(* CoDeSys 2.3 project: cy-wg-06-005.pro *)
(* Title: cy-wg-06 - ClevergyAS *)
(* Author: Andrea Ravasio *)
(* Libraries: Standard.lib 2.12.10 13:48:34, Util.lib*26.9.14 10:12:46, Visual.lib 2.12.10 13:48:34, WagoLibIdent.lib 25.2.13 10:12:16, WagoLibStatus.lib 2.12.10 13:48:32, SysLibFile.lib 2.12.10 13:48:34, SysLibRtc.lib 2.12.10 13:48:32, SysLibSockets.lib 10.2.11 08:20:54, SysLibEvent.lib 2.12.10 13:48:34, SysLibPlcCtrl.lib 2.12.10 13:48:32, SysLibCallback.lib 2.12.10 13:48:32, mod_com.lib 2.12.10 13:48:32, SerComm.lib 31.5.11 07:54:36, Serial_Interface_01.lib 22.4.13 11:50:14, Modb_l05.lib*13.5.15 09:30:08, MBus_03.lib 9.2.13 16:51:58 *)

(* PLC configuration (modules and I/O channels)
K-Bus [K_Bus] node 0, in %IB0 out %QB0
  0750-0402 4 DI 24 V DC 3.0ms [Type_1_4_Channels] node 0, in %IB8 out %QB8 {INTTypePAAssignment = PLC; INTTypeModule = plugged}
    VPN_OUT2 AT %IX4.0 [BOOLOnX_I] Ch_1 Digital input
    KEY_QE_ST AT %IX4.1 [BOOLOnX_I] Ch_2 Digital input
    AT %IX4.2 [BOOLOnX_I] Ch_3 Digital input
    AT %IX4.3 [BOOLOnX_I] Ch_4 Digital input
  0750-0504 4 DO 24V DC 0.5A [Type_10_4_Channels] node 1, in %IB8 out %QB8 {INTTypePAAssignment = PLC; INTTypeModule = plugged}
    AT %QX4.0 [BOOLOnX_Q] Ch_1 Digital output
    AT %QX4.1 [BOOLOnX_Q] Ch_2 Digital output
    TEST1 AT %QX4.2 [BOOLOnX_Q] Ch_3 Digital output
    TEST2 AT %QX4.3 [BOOLOnX_Q] Ch_4 Digital output
  0750-0653/0003-0000#03 RS485 Interface (Adjustable), 3 Bytes [Type_21_1_Channels] node 2, in %IB4 out %QB4 {INTTypePAAssignment = PLC; INTTypeModule = plugged}
    AT %IX0.0 [BOOLOnX_I] Transmission acknowledgement
    AT %IX0.1 [BOOLOnX_I] Reception request
    AT %IX0.2 [BOOLOnX_I] Initialization acknowledgement
    AT %IX0.3 [BOOLOnX_I] Input buffer is full
    AT %IX0.4 [BOOLOnX_I] Number of received characters Bit 0
    AT %IX0.5 [BOOLOnX_I] Number of received characters Bit 1
    AT %IX0.6 [BOOLOnX_I] Number of received characters Bit 2
    AT %IB1 [BYTEOnB_I] Input data Byte 0
    AT %IB2 [BYTEOnB_I] Input data Byte 1
    AT %IB3 [BYTEOnB_I] Input data Byte 2
    AT %QX0.0 [BOOLOnX_Q] Transmission request
    AT %QX0.1 [BOOLOnX_Q] Reception acknowledgement
    AT %QX0.2 [BOOLOnX_Q] Initialization request
    AT %QX0.4 [BOOLOnX_Q] Number of characters Bit 0
    AT %QX0.5 [BOOLOnX_Q] Number of characters Bit 1
    AT %QX0.6 [BOOLOnX_Q] Number of characters Bit 2
    AT %QB1 [BYTEOnB_Q] Output data Byte 0
    AT %QB2 [BYTEOnB_Q] Output data Byte 1
    AT %QB3 [BYTEOnB_Q] Output data Byte 2
  0750-0650/0003-0000#03 RS 232 C Interface (Adjustable), 3 Byte [Type_21_1_Channels] node 0, in %IB4 out %QB4 {INTTypePAAssignment = PLC; INTTypeModule = plugged}
    AT %IX2.0 [BOOLOnX_I] Transmission acknowledgement
    AT %IX2.1 [BOOLOnX_I] Reception request
    AT %IX2.2 [BOOLOnX_I] Initialization acknowledgement
    AT %IX2.3 [BOOLOnX_I] Input buffer is full
    AT %IX2.4 [BOOLOnX_I] Number of received characters Bit 0
    AT %IX2.5 [BOOLOnX_I] Number of received characters Bit 1
    AT %IX2.6 [BOOLOnX_I] Number of received characters Bit 2
    AT %IB5 [BYTEOnB_I] Input data Byte 0
    AT %IB6 [BYTEOnB_I] Input data Byte 1
    AT %IB7 [BYTEOnB_I] Input data Byte 2
    AT %QX2.0 [BOOLOnX_Q] Transmission request
    AT %QX2.1 [BOOLOnX_Q] Reception acknowledgement
    AT %QX2.2 [BOOLOnX_Q] Initialization request
    AT %QX2.4 [BOOLOnX_Q] Number of characters Bit 0
    AT %QX2.5 [BOOLOnX_Q] Number of characters Bit 1
    AT %QX2.6 [BOOLOnX_Q] Number of characters Bit 2
    AT %QB5 [BYTEOnB_Q] Output data Byte 0
    AT %QB6 [BYTEOnB_Q] Output data Byte 1
    AT %QB7 [BYTEOnB_Q] Output data Byte 2
Fieldbus variables [FB_VARS] node 1, in %IB0 out %QB0
Flag variables [FLAG_VARS] node 2, in %IB0 out %QB0
Modbus-Master [MB_MASTER] node 3, in %IB0 out %QB0
*)

(* Global variable list: Global_Constants *)
VAR_GLOBAL CONSTANT

	Plant_NAME			: STRING :='cySN:6 cyVER:5 - Gavazzeni D Energetiche';
	Plant_SN			: DWORD  :=6;  		(* S/N Impianto di telecontrollo *)
	Plant_SW_VER		: WORD   :=5;		(* Versione SW installata *)

	(* Parameters *)
	Plant_DefaultTAmb	: INT	:=100;		(* [.1°C] Temperatura ambiente di default in caso di rottura sonda *)
	Plant_MaxRunTAmb	: INT   :=250; 		(* [.1°C] Temperatura ambiente massima funzionamento impianto *)
	Plant_AntiFreezeTAmb: INT   :=-40;		(* [.1°C] Antifreeze temperature, start circulators *)
	Plant_VRD_TAlarm	: INT   :=450; 		(* [.1°C] Temperatura di allarme VRD, blocco *)
	Plant_VRD_TMax		: INT   :=430; 		(* [.1°C] Setpoint massimo per uscita VRD *)
	Plant_VRD_TDefault	: INT	:=300;		(* [.1°C] Temperatura di default in caso di errore climatica *)
	Plant_CirOffDelay	: TIME	:=T#15m;	(* (Def.T#15m) Ritardo spegnimento pompe per ricircolo caldaia *)
	Plant_MaxWaterLoss	: WORD  :=2;		(* [lt/h] Massima perdita del circuito *)

	(* Filesystem *)
	FilesPath  			: STRING :='S:\';

	(* TCP Logger *)
	Logger_SERVER		: STRING:='';
	Logger_IP			: STRING:='192.168.100.3';
	Logger_PORT			: WORD  :=80;
	Logger_GETSTART		: STRING:='GET /cygmsrv/hsgm.ashx?';
	Logger_GETEND		: STRING:='$R$N$R$N';
	Logger_CHECK		: STRING:='True';
	Logger_CRLF			: STRING:='$R$N';
	Logger_DataFile		: STRING:='S:\LOG.DAT';
	Logger_DataFileOld	: STRING:='S:\LOG.BCK';
	Logger_IndexFile	: STRING:='S:\LOG.IDX';
	Logger_ConnRetries	: BYTE:=5;
	Logger_RecoverMsgs	: BYTE:=25;

	(* TCP Remote *)
	Remote_PORT			: WORD  :=10;
	Remote_WELCOME		: STRING:='Connected$R$N';
	Remote_OK			: STRING:='OK$R$N';
	Remote_ERROR		: STRING:='ERROR$R$N';

	(* TCP Sockets *)
	MAX_SEND_TCP_SERVER					 : DWORD:=1500;(*60000*)
	MAX_RECEIVE_TCP_SERVER				 : DWORD:=3000;
	MAX_RECEIVE_TCP_SERVER_SOCKET	 	 : DWORD:=1500;
	MAX_SEND_TCP_CLIENT					 : DWORD:=1500;(*15000*)
	MAX_RECEIVE_TCP_CLIENT				 : DWORD:=1500;
	MAX_RECEIVE_TCP_CLIENT_SOCKET		 : DWORD:=1500;
	MAX_RECEIVE_UDP_SERVER				 : INT  :=1472;
	MAX_RECEIVE_UDP_CLIENT				 : INT  :=1472;
	CONNECT_WATCHDOG_TIME				 : TIME :=t#10s;

END_VAR

(* Global variable list: Global_Retain *)
VAR_GLOBAL RETAIN PERSISTENT
	Mode_Manual : BOOL := FALSE;
END_VAR

(* Global variable list: Global_Variables *)
VAR_GLOBAL

	SYS    : typ_SYS;

	MODB01 : obj_MODBUS						:= ( ID:=1 , COM:=2, BAUDRATE:=BAUD_9600, RS485:=TRUE );
	GAS02  : obj_MODBUS_ELGAS_MINIELCOR		:= ( ID:=2 , ADDRESS:=1 );

	MBUS01 : obj_MBUS						:= ( ID:=1 , COM:=3, BAUDRATE:=BAUD_2400 );
	CTB05  : obj_MBUS_CTB_SHARKY775			:= ( ID:=5 , ADDRESS:=16#51311890 );
	CTB06  : obj_MBUS_CTB_SHARKY775			:= ( ID:=6 , ADDRESS:=16#51311889 );
	CTB07  : obj_MBUS_CTB_SHARKY775			:= ( ID:=7 , ADDRESS:=16#51038659 );

	Logger : typ_Logger;

	(**** SIMULATION ONLY ****)
(*	VPN_ST2		:BOOL:=TRUE;
	KEY_QE_ST	:BOOL:=TRUE;
*)

END_VAR

(* Data type in Logger *)
TYPE en_Logger_ErrLev :
(
	EL_Log			:=0,
	EL_Wrn			:=1,
	EL_Alarm		:=2,
	EL_AlarmStop	:=3
);
END_TYPE

(* Data type in Logger *)
TYPE en_Logger_Status :
(
	S_Logger_UNKNOWN := 0,
	S_Logger_IDLE,
	S_Logger_WAITCONN,
	S_Logger_WAITTX,
	S_Logger_WAITRESP,
	S_Logger_ERROR
);
END_TYPE

(* Data type *)
TYPE en_SYS_Objects :
(
	EO_SYS		:=0,  (* PLC *)
	EO_VPN		:=1,  (* VPN *)
	EO_DOOR		:=2,  (* Door & access control *)

	EO_CAL		:=10, (* Caldaia *)
	EO_CIR		:=11, (* Circolatore *)
	EO_CRON		:=12, (* Crono-termostato *)
	EO_VRD		:=13, (* Valvola miscelatore pannelli *)
	EO_CTL		:=14, (* Contalitri *)
	EO_CTB		:=15, (* Contabilizzatore *)
	EO_TPV		:=16, (* Temperature probes values *)
	EO_PPV		:=17, (* Pressure probes values *)
	EO_PBV		:=18, (* Over-Pressure Alarms *)
	EO_TBV		:=19, (* Over-Temperature Alarms *)
	EO_PMV		:=20, (* Under-Pressure Alarms *)
	EO_GRU		:=21, (* Gruppo termico *)
	EO_PDC		:=22, (* Pompa di calore *)
	EO_SOL		:=23, (* Pannello solare termico *)
	EO_ESOL		:=24, (* Pannello solare fotovoltaico *)
	EO_GAS		:=25, (* Contatore GAS *)
	EO_PORT		:=26, (* Misuratore di portata *)
	EO_FPV		:=27, (* Flow probes value *)
	EO_ANZ		:=28, (* Analizzatore di rete elettrica *)

	EO_LON		:=1000, (* Bus - LON *)
	EO_MODBUS	:=1001, (* Bus - MODBUS *)
	EO_MBUS		:=1002  (* Bus - M-BUS *)
);
END_TYPE

(* Data type *)
TYPE en_SYS_Status :
(
	S_UNKNOWN  := 0,
	S_STARTUP,
	S_INIT_RTC,
	S_INIT_VAR,
	S_AUTOTEST,
	S_RUNNING,
	S_SHUTDOWN,
	S_HALT
);
END_TYPE

(* Data type in Logger *)
TYPE typ_Logger :
STRUCT
	Status		: en_Logger_Status;

	SendReq		: BOOL;
	SendIdx		: DWORD;
	SendData	: ARRAY [0..MAX_SEND_TCP_CLIENT] OF BYTE;
	SendLen		: DINT;

	TData		: ARRAY [0..MAX_SEND_TCP_CLIENT] OF BYTE;
	TLen		: DINT;

	LastIdxPos	: DWORD;

	(* Temporary variables used by objects *)
	s1			: STRING(256);
	i1			: WORD;

END_STRUCT
END_TYPE

(* Data type in Plant_Objects *)
TYPE typ_MODBUS_ELGAS_MINIELCOR :
STRUCT
	Vb			: ARRAY [0..3] OF WORD;	(* m^3 *)
	Vm			: DWORD;				(* m^3 *)
	P			: REAL;					(* bar *)
	T			: REAL;					(* °C *)
	C			: REAL;
	Vbs			: ARRAY [0..3] OF WORD;	(* m^3 *)
	Vb_d_d		: ARRAY [0..3] OF WORD;	(* m^3 *)
	Vb_d_m		: ARRAY [0..3] OF WORD;	(* m^3 *)
	Vm_d_d		: DWORD;				(* m^3 *)
	Q			: REAL;					(* m^3/h *)
	Qb			: REAL;					(* m^3/h *)

	BC_EVC		: REAL;			(* % *)
	BV_EVC		: REAL;			(* V *)
	D_Err		: WORD;			(* 0:OK, 1:FAIL *)
	Status		: DWORD;		(* Status bits *)

END_STRUCT
END_TYPE

(* Data type in Plant_Objects *)
TYPE typ_MODBUS_VAR : (* Gestione parametri MODBUS *)
STRUCT
	SlaveAddress	: BYTE;
	FunCode			: BYTE;
	FunAddress		: WORD;
	Refresh_Time	: BYTE; (* 0:No refresh x:Refresh in seconds *)
	Refresh_Cnt		: BYTE; (* INTERNAL *)
	Variable		: POINTER TO WORD;
	Variable_Size	: BYTE;
	Variable_Mirror : WORD; (* INTERNAL [Force refresh on read variables when <>0] *)
END_STRUCT
END_TYPE

(* Data type *)
TYPE typ_SYS :
STRUCT
	Status			: en_SYS_Status;
	Warning			: BOOL;
	Alarm			: BOOL;
	AlarmStop		: BOOL;

	Time_LogString	: STRING;
	Time_Year		: WORD;
	Time_Month		: BYTE;
	Time_Day		: BYTE;

	Time_CT_DT		: DT;
	Time_CT_Day		: WORD;
	Time_CT_Quarter	: BYTE;

	LastLogs_Idx	: BYTE;
	LastLogs_Dat	: ARRAY[0..5] OF STRING;
	LastLogs_Msg	: ARRAY[0..5] OF STRING;

END_STRUCT
END_TYPE

(* POU PLC_PRG, ST *)
PROGRAM PLC_PRG
VAR
	Timer1: TON; (* Fast controls tick *)
	Timer2: TON; (* Plant control tick *)
	Timer3: TON; (* Logger timer *)
END_VAR
(******************************************************************************
 ****                           MAIN TASK CODE                             ****
 ******************************************************************************

	Network setup:
		IP  = 192.168.100.2 | MSK = 255.255.255.0
		GW	= 192.168.100.1 | DNS = 192.168.100.1
		SNTP = 193.204.114.232 (3600s) ==> 192.168.100.3

*)

(*==============================*)
(*===== Main status machine ====*)
(*==============================*)
Main_Stm();

(*==============================*)
(*== Running cycle operations ==*)
(*==============================*)
IF SYS.Status>S_INIT_VAR THEN

	(* Execute MODBUS01 process *)
	MODB01();
	GAS02( MODBUS:=MODB01 );

	(* Execute MBUS01 process *)
	MBUS01();
	CTB05( MBUS:=MBUS01 );
	CTB06( MBUS:=MBUS01 );
	CTB07( MBUS:=MBUS01 );

END_IF

(*==============================*)
(*== System cycle operations ===*)
(*==============================*)
(* Execute TCP processes *)
Logger_Proc();
Remote_Proc();
(* Update user led *)
USRLED_Update();
(* Execute Cron Editor commands *)
(*CronEd(); *)
(* External resources *)
(*	IF NOT TPV01.ERR THEN T_AMB:=T_S01;
ELSIF NOT TPV05.ERR THEN T_AMB:=GRU01.TAmb;
ELSE 					 T_AMB:=Plant_DefaultTAmb;
END_IF *)

(**** SIMULATION ONLY ****)
(*...*)
END_PROGRAM
ACTION Main_Stm:
CASE Sys.Status OF

	S_STARTUP:
		Sys.Status:=S_INIT_RTC;

	S_INIT_RTC:
		(* Check RTC and update from network *)
		RTC_Update();
		(* Check time *)
		IF Sys.Time_Year>2000 THEN
			Sys.Status:=S_INIT_VAR;
		END_IF

	S_INIT_VAR:
		LogEv(EL_Wrn,EO_SYS,0,1,CONCAT('System_startup_v',WORD_TO_STRING(Plant_SW_VER)));
		Sys.Status:=S_RUNNING;

	S_RUNNING:
		Timer1(IN:=NOT Timer1.Q,PT:=T#50ms);
		IF Timer1.Q THEN
			(* Update meters *)

			(* Update system checks *)
			SYS_Proc();
		END_IF

		Timer2(IN:=NOT Timer2.Q,PT:=T#500ms);
		IF Timer2.Q THEN
			(* Read current date/time *)
			RTC_Update();
			(* Execute plant operations *)

			(* Test toggle *)
			IF TEST1 THEN TEST1:=FALSE; ELSE TEST1:=TRUE; END_IF
		END_IF

		Timer3(IN:=NOT Timer3.Q,PT:=T#5m);
		IF Timer3.Q THEN
			(* Trig logger *)
			LogTrig();
			(* Execute temporary CSV logger *)
			(*CSV_Log();*)
		END_IF

	S_SHUTDOWN:
		(* Stop sistema *)
		Sys.Status:=S_STARTUP;

	S_HALT:
		(* Aspetta uscita manuale *)
		Sys.Status:=S_STARTUP;

ELSE
	Sys.Status:=S_STARTUP;
END_CASE;
END_ACTION

(* POU TCP_Logger/Logger_Proc, ST *)
PROGRAM Logger_Proc
VAR
	c1:         	TCPCLIENT;

	Open:	    	BOOL;
	IpAddr:			DWORD;
	InetAddr:		DWORD;
	Connected:  	BOOL;
	Error:      	DINT;
	TxTrig:     	BOOL;
	RxData:			ARRAY [0..MAX_RECEIVE_TCP_CLIENT] OF BYTE;
	RxLen:			DINT;

	Retry:			BYTE;	(* Counter for connection retries *)
	Recovered:		BYTE;	(* Counter for recovered unsent messages *)

	i:				DINT;
	pos:			DWORD;
	hFile:			DWORD;

END_VAR
(*=== State machine ===*)
CASE Logger.Status OF

	S_Logger_UNKNOWN:
		(* Startup *)
		Logger.SendReq:=FALSE;
		Open:=FALSE;
		Logger.Status:=S_Logger_IDLE;

	S_Logger_IDLE:
		(* Wait request *)
		IF Logger.SendReq THEN
			(* Resolve server name or use static IP *)
			IF LEN(Logger_SERVER)=0 THEN
				InetAddr:=SysSockInetAddr(Logger_IP);
			ELSE
				IpAddr:=SysSockGetHostByName(ADR(Logger_SERVER));
				DWORDSWAP(pIn:=ADR(IpAddr), pOut:=ADR(InetAddr));
			END_IF
			TxTrig:=FALSE;
			RxLen:=0;
			(* Open connection *)
			Open:=TRUE;
			Logger.Status:=S_Logger_WAITCONN;
		END_IF

	S_Logger_WAITCONN:
		(* Wait connection *)
		IF Connected THEN
			(* Send data *)
			TxTrig:=TRUE;
			Logger.Status:=S_Logger_WAITTX;
		END_IF
		IF Error>0 THEN
			Open:=FALSE;
			Logger.Status:=S_Logger_ERROR;
		END_IF

	S_Logger_WAITTX:
		(* Wait transmission *)
		IF NOT TxTrig THEN
			Logger.Status:=S_Logger_WAITRESP;
		END_IF
		IF Error>0 THEN
			Open:=FALSE;
			Logger.Status:=S_Logger_ERROR;
		END_IF

	S_Logger_WAITRESP:
		(* Wait response *)
		IF Connected=FALSE (* OR TIMEOUT!! *) THEN
			Open:=FALSE;
			(* Check response *)
			IF RxLen>=4 AND CHKSTRING(pString:=ADR(RxData), pPattern:=ADR(Logger_CHECK)) THEN
				Logger.SendReq:=FALSE;
				Retry:=0;
				(* Check unsent messages to flush *)
				IF Recovered<Logger_RecoverMsgs THEN
					MsgChk();
					IF Logger.SendReq=TRUE THEN
						Recovered:=Recovered+1;
					ELSE
						Recovered:=0;
					END_IF
				ELSE
					Recovered:=0;
				END_IF
				Logger.Status:=S_Logger_IDLE;
			ELSE
				Logger.Status:=S_Logger_ERROR;
			END_IF
		END_IF

	S_Logger_ERROR:
		(* Connection error or send failure *)
		Retry:=Retry+1;
		IF Retry>Logger_ConnRetries THEN
			(* Save message as unsent *)
			MsgSave();
			Logger.SendReq:=FALSE;
			Retry:=0;
		END_IF
		Logger.Status:=S_Logger_IDLE;

ELSE
	Logger.Status:=S_Logger_UNKNOWN;
END_CASE


(*=== Execute client lib ===*)
c1(
	xOpenConnection			:= Open,
	dwInetAddr 				:= InetAddr,
	wPortNumber				:= Logger_PORT,
	ptSendData				:= ADR(Logger.SendData),
	diSendCount				:= Logger.SendLen,
	tConnectWatchdogTime	:= t#10s,
	xStartSend				:= TxTrig,
	aReceiveBuffer			:= RxData,
	diReceiveCount			:= RxLen,
	xConnected				=> Connected,
	diError					=> Error
);

(*=== Process Rx data ===*)
(*IF RxLen>0 THEN
	RxLen:=0;
END_IF*)
END_PROGRAM
ACTION MsgChk:
(* Open index file *)
hFile:=SysFileOpen(Logger_IndexFile,'r');
IF hFile=0 THEN
	RETURN;
END_IF
(* Search oldest message to recover *)
SysFileSetPos(hFile,Logger.LastIdxPos);
Logger.SendLen:=0;
REPEAT
	SysFileRead(hFile, ADR(Logger.SendIdx), SIZEOF(Logger.SendIdx));
	pos:=SysFileGetPos(hFile);
	SysFileRead(hFile, ADR(Logger.SendLen), SIZEOF(Logger.SendLen));
UNTIL
	SysFileEOF(hFile) OR Logger.SendLen<>0
END_REPEAT
SysFileClose(hFile);
(* Delete index file when all messages are recovered *)
IF Logger.SendLen=0 THEN
	Logger.LastIdxPos:=0;
	SysFileDelete(Logger_IndexFile);
	RETURN;
END_IF
(* Recover message data *)
hFile:=SysFileOpen(Logger_DataFile,'r');
IF hFile<>0 THEN
	SysFileSetPos(hFile,Logger.SendIdx);
	SysFileRead(hFile,ADR(Logger.SendData),Logger.SendLen);
	Logger.SendReq:=TRUE;
	SysFileClose(hFile);
END_IF
(* Clear index entry *)
hFile:=SysFileOpen(Logger_IndexFile,'a');
IF hFile<>0 THEN
	SysFileSetPos(hFile,pos);
	i:=0;
	SysFileWrite(hFile, ADR(i), 4);
	Logger.LastIdxPos:=SysFileGetPos(hFile);
	SysFileClose(hFile);
END_IF
END_ACTION
ACTION MsgSave:
(* Add log position in recovery indexes *)
hFile:=SysFileOpen(Logger_IndexFile,'a');
SysFileWrite(hFile, ADR(Logger.SendIdx), SIZEOF(Logger.SendIdx));
SysFileWrite(hFile, ADR(Logger.SendLen), SIZEOF(Logger.SendLen));
SysFileClose(hFile);
END_ACTION

(* POU Utils Functions/TCPCLIENT, ST *)
FUNCTION_BLOCK TCPCLIENT
(***********************************************************************************************************	*)
(* Version: 1.3b                        			          													*)
(* Date: 28.10.2014                   				          							            			*)
(***********************************************************************************************************	*)
(* WAGO Kontakttechnik GmbH Hansastr. 27 32423 Minden(Westf.)													*)
(* Tel. +0049 571/887-0 Fax. +0049 571/887-0																	*)
(* Author: VB																									*)
(***********************************************************************************************************	*)
(*Description:	A TCP client to read and write data with additional connection watchdog							*)
(*History:																										*)
(*Version 1.3b: 28.10.2014: Use DWORD address for IP (Andrea Ravasio)											*)
(*Version 1.3: 11.02.2011: Changes according to 750-880/881											 			*)
(*Version 1.2: 29.08.2007 Bugfix TCP Client																		*)
(*Version 1.1: 15.01.2007 Changes according to FW11																*)
(*Version 1.0: 09.03.2006 Release																				*)
(***********************************************************************************************************	*)
VAR CONSTANT
	STATE_CREATE     				 : BYTE:= 0;
	STATE_OPEN     					 : BYTE:= 1;
	STATE_IOCTL    					 : BYTE:= 2;
	STATE_CONNECT     				 : BYTE:= 10;
	STATE_TX       					 : BYTE:= 20;
	STATE_RX       					 : BYTE:= 30;
	STATE_CLOSE    					 : BYTE:= 40;
	STATE_ERROR_TRAP			     : BYTE:= 200;
END_VAR

VAR_INPUT
	xOpenConnection					: BOOL;
	dwInetAddr						: DWORD; (* <== Use SysSockInetAddr() value or
													swapped bytes order of SysSockGetHostByName() value *)
	wPortNumber						: WORD;
	ptSendData						: POINTER TO ARRAY[0..MAX_SEND_TCP_CLIENT] OF BYTE;
	diSendCount						: DINT;
	tConnectWatchdogTime		    : TIME := t#10s;
END_VAR
VAR_OUTPUT
	xConnected						: BOOL;
	diError 						: DINT := 0;
END_VAR
(* ErrorCodes -----------------------------------------
	16#8001 => No socket descriptor available 
	16#8002 => SysSockSend returns -1 
	16#8003 => Socket was "gracefully closed" 
	16#8004 => switching to none blocking mode fails
	16#8005 => SysSockClose() returns FALSE 
    16#8006 => SysSockConnect() fails
    16#8007 => SysSockSend() fails
	16#8008 => error state machine 
	16#8009 => timeout while waiting for data from server 
------------------------------------------------------------*)
VAR_IN_OUT
	xStartSend							: BOOL;
	aReceiveBuffer						: ARRAY [0..MAX_RECEIVE_TCP_CLIENT] OF BYTE;
	diReceiveCount						: DINT;
END_VAR
VAR
	m_State								: BYTE := 0;
	m_ReceiveBuffer						: ARRAY [0..MAX_RECEIVE_TCP_CLIENT_SOCKET] OF BYTE;
	m_Socket							: DINT;
	m_AddressInfo						: SOCKADDRESS;
	m_BytesReceived						: DINT;
	m_diReturn							: DINT;
	m_xReturn							: BOOL;
	m_IoCtlParameter  					: DINT := 1; (* IOCTL-Parameter for non-blocking mode of sockets *)
	i									: INT;
	T_Connect							: TON;
	m_count								: DINT;
	diOption							: DINT := 1;
	m_Blocking   						: DINT := 0;
END_VAR
IF xOpenConnection THEN
	(* State maschine *)
	CASE  m_State OF

	(* -------------------------------------------------------------------------*)
	STATE_CREATE:
			(* create socket descriptor*)
			m_Socket := SysSockCreate(diAddressFamily	:= SOCKET_AF_INET,
													 diType		:= SOCKET_STREAM,
													 diProtocol := SOCKET_IPPROTO_TCP);
			IF m_Socket >= 0 THEN
			(*Set Push-Bit*)
				IF ADR(%MW0)=16#30000000  OR ADR(%MW0)=16#20000000 THEN (*841 or 881*)
					SysSockSetOption(
						diSocket:=m_Socket,
						diLevel:=6,
						diOption:=SOCKET_TCP_NODELAY,
						pOptionValue:=ADR(diOption),
						diOptionLength:=SIZEOF(diOption));
				ELSE
						;
				END_IF
				m_State := STATE_IOCTL; (* succesful *)
			ELSE
				diError := 16#8001;  (* no socket descriptor available *)
				m_State := STATE_ERROR_TRAP;
			END_IF

	(* -------------------------------------------------------------------------*)
	STATE_IOCTL: (* change  socket mode  to none blocking *)
		m_diReturn := SysSockIoctl( m_Socket, SOCKET_FIONBIO, ADR(m_IoCtlParameter));
		IF m_diReturn <> 0 THEN
			m_AddressInfo.sin_family := SOCKET_AF_INET;
			m_AddressInfo.sin_port := SysSockNtohs(wPortNumber);
			m_AddressInfo.sin_addr := dwInetAddr;
			m_State := STATE_CONNECT;
		ELSE
			diError := 16#8004;  (* switching to none blocking mode fails *)
			m_State := STATE_ERROR_TRAP;
		END_IF


	(* -------------------------------------------------------------------------*)
	STATE_CONNECT: (* connect with server *)
		T_Connect(IN:=TRUE , PT:=tConnectWatchdogTime);(*activate watchdog for establishing connection to a server*)
		m_xReturn := SysSockConnect ( m_Socket, ADR(m_AddressInfo),  SIZEOF(m_AddressInfo));
		IF m_xReturn THEN (* succesful *)
			IF xStartSend THEN
				m_State := STATE_TX;(*transmit data*)
			ELSE
				m_State := STATE_RX;(*wait for data from server*)
			END_IF
			xConnected:=TRUE;
			T_Connect(IN:=FALSE);
		ELSE
			IF T_Connect.Q THEN
				diError := 16#8006;  (* connect fails *)
				xConnected:=FALSE;
				T_Connect(IN:=FALSE);
				m_State := STATE_ERROR_TRAP;
				SysSockClose( m_Socket);
			ELSE
				m_State := STATE_CONNECT;(*client still  tries to set up connection*)
			END_IF
		END_IF


	STATE_TX:	 (* send TCP-message *)
		m_diReturn := SysSockSend(diSocket := m_Socket,
								  pbyBuffer := ADR(ptSendData^[0]),
								  diBufferSize := diSendCount-m_count,
								  diFlags := 0);

		CASE m_diReturn OF
		-1:	(* ERROR *)
			T_Connect(IN:=TRUE , PT:=CONNECT_WATCHDOG_TIME);(*activate watchdog to check communication*)
			IF t_Connect.Q THEN
				diError := 16#8007;
				T_Connect(IN:=FALSE);
				m_State:=STATE_CLOSE;
			END_IF
		0: (* socket was "gracefully closed" *)
			m_State := STATE_CLOSE;
			diError := 16#8003;
		ELSE (* succesful *)
			m_count:=m_count+m_diReturn;
			IF m_count>=diSendCount THEN
				diError := 16#0000;
				m_State := STATE_RX;
				m_count:=0;
				xStartSend:=FALSE;
			END_IF
			T_Connect(IN:=FALSE);
		END_CASE

	(* -------------------------------------------------------------------------*)
	STATE_RX: (* process receive data *)
			m_BytesReceived := SysSockRecv(	diSocket 	:= m_Socket,
										pbyBuffer 	:= ADR(m_ReceiveBuffer),		(* Address of receive buffer *)
										diBufferSize:= SIZEOF(m_ReceiveBuffer),
										diFlags		:= 0);

			CASE m_BytesReceived OF
			-1:	(* No data available or error occured *)
				T_Connect(IN:=TRUE , PT:=tConnectWatchdogTime);(*activate watchdog to check communication*)
				IF t_Connect.Q THEN
					diError:=16#8009;
					T_Connect(IN:=FALSE);
					m_State:=STATE_CLOSE;
				END_IF
				IF xStartSend THEN
					m_State:=STATE_TX	;(* WAIT IN THIS STATE  and check for arriving data or new send command*)
				END_IF;
			0: (* socket was "gracefully closed"  *)
				m_State:=STATE_CLOSE;
				diError := 16#8003;
			ELSE (* succesful *)
				diError := 16#0000;
				T_Connect(IN:=FALSE);
				(* Copy received data into receive buffer *)
				FOR i:= 0 TO DINT_TO_INT(m_BytesReceived	)-1 DO
					aReceiveBuffer[diReceiveCount]:= m_ReceiveBuffer[i];
					diReceiveCount:=(diReceiveCount+1) MOD SIZEOF(aReceiveBuffer);
				END_FOR

			END_CASE

	(* -------------------------------------------------------------------------*)
	STATE_CLOSE : (* close socket *)
		IF ADR(%MW0)=16#30000000  OR ADR(%MW0)=16#20000000 THEN (*841 or 881*)
			;
		ELSE
			SysSockShutdown(m_Socket, 0);;(*870*)
		END_IF
		m_xReturn := SysSockClose( m_Socket);
		m_Socket := -1;
		m_State := 0; (* succesful *)
		xConnected:=FALSE;
		T_Connect(IN:=FALSE);
	(* -------------------------------------------------------------------------*)
	STATE_ERROR_TRAP: (* error handling *)
		xConnected:=FALSE;

	ELSE  (* Bad FSM code trap  *)
			m_State:= STATE_ERROR_TRAP;
			diError:= 16#8008;
	END_CASE

ELSE(*close connection*)
	IF m_Socket >= 0 THEN
		IF ADR(%MW0)=16#30000000  OR ADR(%MW0)=16#20000000 THEN (*841 or 881*)
			;
		ELSE
			SysSockShutdown(m_Socket, 0);;(*870*)
		END_IF
		SysSockClose( m_Socket);
	END_IF
	m_Socket := -1;
	diError := 16#0000;
	m_State := STATE_CREATE;
	xConnected:=FALSE;
	T_Connect(IN:=FALSE);
END_IF
END_FUNCTION_BLOCK

(* POU Utils Functions/DWORDSWAP, ST *)
FUNCTION DWORDSWAP:BOOL
VAR_INPUT
	pIn:POINTER TO ARRAY[1..4] OF BYTE;
	pOut:POINTER TO ARRAY[1..4] OF BYTE;
END_VAR
VAR
END_VAR
pOut^[1]:=pIn^[4];
pOut^[2]:=pIn^[3];
pOut^[3]:=pIn^[2];
pOut^[4]:=pIn^[1];
END_FUNCTION

(* POU Utils Functions/CHKSTRING, ST *)
FUNCTION CHKSTRING : BOOL
VAR_INPUT
	pString: POINTER TO BYTE;
	pPattern: POINTER TO BYTE;
END_VAR
VAR
END_VAR
CHKSTRING:=TRUE;
WHILE pPattern^<>0 AND CHKSTRING DO
	IF pPattern^<>pString^ THEN CHKSTRING:=FALSE; END_IF
	pString:=pString+1;
	pPattern:=pPattern+1;
END_WHILE
END_FUNCTION

(* POU TCP_Remote/Remote_Proc, ST *)
PROGRAM Remote_Proc
VAR
	s1:         	TCPSERVER;
	Enable: 		BOOL;
	Connected: 		BOOL;
	Error: 			DINT;

	TxData:			ARRAY [0..MAX_SEND_TCP_SERVER] OF BYTE;
	TxLen:			DINT;
	TxTrig:			BOOL;

	RxData:			ARRAY [0..MAX_RECEIVE_TCP_SERVER] OF BYTE;
	RxLen:			DINT;

	Status:			DINT;

	(* Command interpreter *)

	Cmd_Buf:		ARRAY [0..MAX_RECEIVE_TCP_SERVER] OF BYTE;
	Cmd_Buf_U16:	POINTER TO WORD;
	Cmd_Buf_INT:	POINTER TO INT;
	Cmd_BufLen:		WORD;
	Cmd_St:			WORD;

	Cmd_Obj:		WORD;
	Cmd_ObjIdx:		WORD;
	Cmd_C:			WORD;
	Cmd_R:			WORD;
	Cmd_CLen:		WORD;
	Cmd_RLen:		WORD;

	i : WORD;
	j : INT;
	s2 : STRING;

	(* per aggiornare la data e l'ora *)
	SetAnno: INT;
	SetMese: INT;
	SetGiorno: INT;
	SetOra: INT;
	SetMinuti: INT;
	SetSecondi: INT;

END_VAR
(*=== State machine ===*)
CASE Status OF
	0: (* Startup *)
		TxLen:=0; TxTrig:=FALSE;
		RxLen:=0;
		Enable:=TRUE;
		Status:=1;

	1: (* Wait incoming connection *)
		IF Connected THEN
			(* Log access *)
			LogEv(EL_Log,EO_VPN,1,5,'Remote');
			(* Send welcome message *)
			ADDSTRING(pTxData:=ADR(TxData), pString:=ADR(Remote_WELCOME), TxLen:=TxLen);
			TxTrig:=TRUE;
			(* Reset vars *)
			Cmd_BufLen:=0;
			Cmd_St:=0;
			Status:=2;
		END_IF
		IF Error>1 THEN
			Enable:=FALSE;
			Status:=0;
		END_IF

	2: (* Wait command *)
		IF RxLen>0 THEN
			(*=== Interpreter start ===*)
			IF Cmd_BufLen+(RxLen/2)>=MAX_RECEIVE_TCP_SERVER THEN
				(* ERROR *)
				Cmd_BufLen:=0;
			ELSE
				i:=HEXTORAW(pString:=ADR(RxData), StringLen:=DINT_TO_WORD(RxLen), pData:=ADR(Cmd_Buf[Cmd_BufLen]));
				Cmd_BufLen:=Cmd_BufLen+i;
			END_IF
			IF Cmd_BufLen>=8 THEN
				Cmd_Buf_U16:=ADR(Cmd_Buf[6]);
				IF Cmd_BufLen>=(8+Cmd_Buf_U16^) THEN
					Cmd_CLen:=Cmd_Buf_U16^;
					Cmd_Buf_U16:=ADR(Cmd_Buf[0]); Cmd_Obj:=Cmd_Buf_U16^;
					Cmd_Buf_U16:=ADR(Cmd_Buf[2]); Cmd_ObjIdx:=Cmd_Buf_U16^;
					Cmd_Buf_U16:=ADR(Cmd_Buf[4]); Cmd_C:=Cmd_Buf_U16^;

					s2:='RCmd_';		s2:=CONCAT(s2,WORD_TO_STRING(Cmd_Obj));
					s2:=CONCAT(s2,'_'); s2:=CONCAT(s2,WORD_TO_STRING(Cmd_ObjIdx));
					s2:=CONCAT(s2,'_'); s2:=CONCAT(s2,WORD_TO_STRING(Cmd_C));
					s2:=CONCAT(s2,'_');	s2:=CONCAT(s2,WORD_TO_STRING(Cmd_CLen));
					LogEv(EL_Log,EO_VPN,1,6,s2);

					Command();
					Cmd_BufLen:=0;
				END_IF
			END_IF
			(*=== Interpreter end ===*)
			RxLen:=0;
		END_IF
		IF NOT Connected THEN
			Status:=0;
		END_IF

ELSE
	Status:=0;
END_CASE


(*=== Execute server lib ===*)
s1(
	xEnable				:= Enable,
	wPortNumber			:= Remote_PORT,
	tServerTimeOut		:= t#15m,
	ptSendData			:= ADR(TxData),
	diSendCount			:= TxLen,
	xStartSend			:= TxTrig,
	aReceiveBuffer		:= RxData,
	diReceiveCount		:= RxLen,
	xClientConnected	=> Connected,
	diError				=> Error
);
END_PROGRAM
ACTION Cmd_CAL:
(* Check index *)(*
IF Cmd_ObjIdx<1 OR Cmd_ObjIdx>2 THEN
	Cmd_R:=2;
	RETURN;
END_IF

(* Process command *)
CASE Cmd_C OF

	3: (* TRY REARM *)
		IF Cmd_ObjIdx=1 THEN
			CAL01.Rearm:=TRUE;
		ELSE
			CAL02.Rearm:=TRUE;
		END_IF

ELSE
	Cmd_R:=3;
END_CASE
*);
END_ACTION
ACTION Cmd_CRON:
(* Check index *)(*
IF Cmd_ObjIdx<1 OR Cmd_Obj=2 OR Cmd_ObjIdx>6 THEN
	Cmd_R:=2;
	RETURN;
END_IF

(* Process command *)
CASE Cmd_C OF

	1: (* GET PROFILE *)
		IF Cmd_CLen<>3 THEN
			Cmd_R:=4;
		ELSE
			(* Load profile *)
			CronEd.CN_Sel:=WORD_TO_BYTE(Cmd_ObjIdx);
			Cmd_Buf_U16:=ADR(Cmd_Buf[8]);
			CronEd.CN_YSel:=Cmd_Buf_U16^;
			CronEd.PR_Sel:=Cmd_Buf[10];
			CronEd.PR_Load_Exe();
			(* Copy data *)
			Cmd_RLen:=192;
			TxLen:=TxLen+RAWTOHEX(ADR(CronEd.PR.Setpoint),192,ADR(TxData[TxLen]));
		END_IF

	2: (* SET PROFILE *)
		IF Cmd_CLen<>(3+192) THEN
			Cmd_R:=4;
		ELSE
			(* Save profile *)
			CronEd.CN_Sel:=WORD_TO_BYTE(Cmd_ObjIdx);
			Cmd_Buf_U16:=ADR(Cmd_Buf[8]);
			CronEd.CN_YSel:=Cmd_Buf_U16^;
			CronEd.PR_Sel:=Cmd_Buf[10];
			MEMCPY(ADR(Cmd_Buf[11]),ADR(CronEd.PR.Setpoint),192);
			CronEd.PR_Save_Exe();
		END_IF

	5: (* GET CALENDAR MONTH *)
		IF Cmd_CLen<>3 THEN
			Cmd_R:=4;
		ELSE
			(* Load calendar *)
			CronEd.CN_Sel:=WORD_TO_BYTE(Cmd_ObjIdx);
			Cmd_Buf_U16:=ADR(Cmd_Buf[8]);
			CronEd.CN_YSel:=Cmd_Buf_U16^;
			CronEd.CA_Sel:=Cmd_Buf[10];
			CronEd.CA_Load_Exe();
			(* Copy data *)
			Cmd_RLen:=32;
			TxLen:=TxLen+RAWTOHEX(ADR(CronEd.CA.Profile),32,ADR(TxData[TxLen]));
		END_IF

	6: (* SET CALENDAR MONTH *)
		IF Cmd_CLen<>(3+32) THEN
			Cmd_R:=4;
		ELSE
			(* Save calendar *)
			CronEd.CN_Sel:=WORD_TO_BYTE(Cmd_ObjIdx);
			Cmd_Buf_U16:=ADR(Cmd_Buf[8]);
			CronEd.CN_YSel:=Cmd_Buf_U16^;
			CronEd.CA_Sel:=Cmd_Buf[10];
			MEMCPY(ADR(Cmd_Buf[11]),ADR(CronEd.CA.Profile),32);
			CronEd.CA_Save_Exe();
		END_IF

ELSE
	Cmd_R:=3;
END_CASE
*);
END_ACTION
ACTION Cmd_GRU:
(* Check index *)(*
IF Cmd_ObjIdx<>1 THEN
	Cmd_R:=2;
	RETURN;
END_IF

(* Process command *)
CASE Cmd_C OF

	1: (* GET CLIMATIC *)
		Cmd_RLen:=20;
		FOR i:=0 TO 4 DO
			j:=DINT_TO_INT(GRU01_Clima.Points[i].X);
			TxLen:=TxLen+RAWTOHEX(ADR(j),2,ADR(TxData[TxLen]));
			j:=DINT_TO_INT(GRU01_Clima.Points[i].Y);
			TxLen:=TxLen+RAWTOHEX(ADR(j),2,ADR(TxData[TxLen]));
		END_FOR

	2: (* SET CLIMATIC *)
		IF Cmd_CLen<>20 THEN
			Cmd_R:=4;
		ELSE
			FOR i:=0 TO 4 DO
				Cmd_Buf_INT:=ADR(Cmd_Buf[8+4*i]); j:=Cmd_Buf_INT^;
				GRU01_Clima.Points[i].X:=INT_TO_DINT(j);
				Cmd_Buf_INT:=ADR(Cmd_Buf[10+4*i]); j:=Cmd_Buf_INT^;
				GRU01_Clima.Points[i].Y:=INT_TO_DINT(j);
			END_FOR
		END_IF

ELSE
	Cmd_R:=3;
END_CASE
*);
END_ACTION
ACTION Cmd_PDC:
;(* Check index *)(*
IF Cmd_ObjIdx<>1 THEN
	Cmd_R:=2;
	RETURN;
END_IF

(* Process command *)
CASE Cmd_C OF

	3: (* TRY REARM *)
		PDC01.Rearm:=TRUE;

ELSE
	Cmd_R:=3;
END_CASE
*);
END_ACTION
ACTION Cmd_SYS:
(* Check index *)
IF Cmd_ObjIdx<>0 THEN
	Cmd_R:=2;
	RETURN;
END_IF

(* Process command *)
CASE Cmd_C OF

	0: (* ECHO *)
		IF Cmd_CLen<>0 THEN
			TxLen:=0;
		END_IF

	1: (* LOG REQUEST *)
		LogTrig();

	2: (* REARM *)
		Sys.Warning:=FALSE;
		Sys.Alarm:=FALSE;
		Sys.AlarmStop:=FALSE;
		MODB01.VARS_Alarm:=FALSE;

	3: (* GET INFO1 *)
		Cmd_RLen:=6;
		TxLen:=TxLen+RAWTOHEX(ADR(Plant_SN),4,ADR(TxData[TxLen]));
		TxLen:=TxLen+RAWTOHEX(ADR(Plant_SW_VER),2,ADR(TxData[TxLen]));

	14: (*  Imposto data e ora del PLC  *)


			Cmd_Buf_U16:=ADR(Cmd_Buf[8]);
			SetAnno:= Cmd_Buf_U16^; 												(* Anno *)
			Cmd_Buf_U16:=ADR(Cmd_Buf[10]);
			SetMese:= Cmd_Buf_U16^;												 	(* mese *)
			Cmd_Buf_U16:=ADR(Cmd_Buf[12]);
			SetGiorno:=( Cmd_Buf_U16^);											 	(* Giorno *)
			Cmd_Buf_U16:=ADR(Cmd_Buf[14]);
			SetOra:=( Cmd_Buf_U16^); 												(* ora *)
			Cmd_Buf_U16:=ADR(Cmd_Buf[16]);
			SetMinuti:= ( Cmd_Buf_U16^);										 	(* Minuti *)
			Cmd_Buf_U16:=ADR(Cmd_Buf[18]);
			SetSecondi:= ( Cmd_Buf_U16^);										 	(* secondi *)

			SysRtcSetTime((SetDataTime(SetAnno,SetMese,SetGiorno,SetOra,SetMinuti,SetSecondi)));



ELSE
	Cmd_R:=3;
END_CASE
END_ACTION
ACTION Command:
(* Default response OK/NODATA *)
Cmd_R:=0;
Cmd_RLen:=0;
TxLen:=16;

(* Check object *)
CASE Cmd_Obj OF

	EO_SYS:
		Cmd_SYS();
(*
	EO_GRU:
		Cmd_GRU();

	EO_PDC:
		Cmd_PDC();

	EO_CAL:
		Cmd_CAL();

	EO_CRON:
		Cmd_CRON();
*)
ELSE
	Cmd_R:=1;
END_CASE

(* Generate response *)
IF TxLen>0 THEN
	RAWTOHEX(ADR(Cmd_Obj)	,2,ADR(TxData[ 0]));
	RAWTOHEX(ADR(Cmd_ObjIdx),2,ADR(TxData[ 4]));
	RAWTOHEX(ADR(Cmd_R)		,2,ADR(TxData[ 8]));
	RAWTOHEX(ADR(Cmd_RLen)	,2,ADR(TxData[12]));
	TxTrig:=TRUE;
END_IF
END_ACTION

(* POU Utils Functions/TCPSERVER, ST *)
FUNCTION_BLOCK TCPSERVER
(***********************************************************************************************************	*)
(* Version: 1.6                                    			          											*)
(* Date: 11.02.2011                                   					          							    *)
(***********************************************************************************************************	*)
(* WAGO Kontakttechnik GmbH Hansastr. 27 32423 Minden(Westf.)													*)
(* Tel. +0049 571/887-0 Fax. +0049 571/887-0																	*)
(* Author: VB																									*)
(***********************************************************************************************************	*)
(*Description:	A TCP server to read and write data													       		*)
(*Historie:																										*)
(*Version 1.6: 11.02.2011: Changes according to 750-880/881											 			*)
(*Version 1.5: 27.11.2008 Bugfix allow reuse port																*)
(*Version 1.4: 13.10.2008 Bugfix transmitting large data														*)
(*Version 1.3: 15.01.2007 Changes according to FW11																*)
(*Version 1.2: 09.03.2006 Changes for socket handle 0											       			*)
(*Version 1.1: 14.02.2005 Release																				*)
(***********************************************************************************************************	*)
VAR CONSTANT
	STATE_INIT     				 : BYTE:= 0;
	STATE_OPEN     				 : BYTE:= 1;
	STATE_TX       				 : BYTE:= 20;
	STATE_RX       				 : BYTE:= 30;
	STATE_CLOSE    				 : BYTE:= 40;
	STATE_ERROR_TRAP		 	 : BYTE:= 200;
END_VAR
VAR_INPUT
	xEnable    					: BOOL;	 (* Set TRUE to enable function block *)
	wPortNumber					: WORD;  (* Port *)
	tServerTimeOut				: TIME:=t#50s;
	ptSendData					: POINTER TO ARRAY[0..MAX_SEND_TCP_SERVER] OF BYTE;
	diSendCount					: DINT;
END_VAR
VAR_OUTPUT
	xClientConnected  			: BOOL:= FALSE;
	diError 					: DINT:= 0;
END_VAR
(* Status Codes -----------------------------------------
	16#8001 => No socket descriptor available 
	16#8002 => SysSockBind fails 
	16#8003 => SysSockListen fails 
	16#8004 => switching to none blocking mode fails
	16#8005 => SysSockClose() returns FALSE 
    16#8006 => SysSockConnect() fails
    16#8007 => SysSockSend() fails
	16#8008 => error state machine 
	16#8009 => timeout while waiting for data from server 
	16#0001 => server waiting for client to establish connection
------------------------------------------------------------*)
VAR_IN_OUT
	xStartSend					: BOOL;
	aReceiveBuffer				: ARRAY [0..MAX_RECEIVE_TCP_SERVER] OF BYTE;
	diReceiveCount				: DINT;
END_VAR

VAR
	m_State    					: BYTE:= 0;
	m_ReceiveBuffer				: ARRAY [0..MAX_RECEIVE_TCP_SERVER_SOCKET] OF BYTE;
	m_ServerSocket				: DINT:= SOCKET_INVALID;
	m_Socket					: DINT:= SOCKET_INVALID;
	m_AddressInfo				: SOCKADDRESS;
	m_BytesReceived				: DINT;
	m_diReturn					: DINT;
	m_xReturn					: BOOL;
	m_SizeSockadr				: DWORD;
	m_ConnectionWatchdog		: TON;
	m_Flags						: DINT;
	m_NoneBlocking   			: DINT:= 1;
	m_Blocking   				: DINT:= 0;
	i							: INT;
	m_count						: DINT;
	diOption					: DINT := 1;
	on: DINT;
END_VAR
IF xEnable THEN
	CASE m_State OF
		STATE_INIT:
			(* Create Socket *)
			m_ServerSocket:= SysSockCreate( SOCKET_AF_INET, SOCKET_STREAM, 0);
			IF m_ServerSocket = SOCKET_INVALID THEN
				(* *)
				diError:= 16#8001;
				m_State:= STATE_ERROR_TRAP;
				RETURN;
			ELSE
				;
			END_IF
			(* Address bindings *)
			(********************)
			on:=1;
			SysSockSetOption( m_ServerSocket, SOCKET_SOL, SOCKET_SO_REUSEADDR, ADR(on), SIZEOF(on) );

			m_AddressInfo.sin_family:= SOCKET_AF_INET;
			m_AddressInfo.sin_port  := SysSockHtons( wPortNumber);
			m_AddressInfo.sin_addr  := SOCKET_INADDR_ANY;
			IF NOT SysSockBind( m_ServerSocket, ADR(m_AddressInfo), SIZEOF(m_AddressInfo)) THEN
				diError:= 16#8002;
				m_State:= STATE_ERROR_TRAP;
				RETURN;
			END_IF
			(* Wait for connections *)
			(************************)
			IF NOT SysSockListen( m_ServerSocket, 1) THEN
				diError:= 16#8003;
				m_State:= STATE_ERROR_TRAP;
			END_IF

			(* Puts SOCKET in NonBlocking mode *)
			m_diReturn:= SysSockIoctl( m_ServerSocket, SOCKET_FIONBIO, ADR(m_NoneBlocking));

			m_State:= STATE_OPEN;


		STATE_OPEN: 	(* Waiting for incomming connection *)
				m_SizeSockadr:=SIZEOF(m_AddressInfo);
				m_Socket:= SysSockAccept( m_ServerSocket, ADR(m_AddressInfo), ADR(m_SizeSockadr));
				diError:=State_open;
				IF m_Socket <> SOCKET_INVALID THEN
					xClientConnected:=TRUE;
					(*Set Push-Bit:new V1.5*)
					IF ADR(%MW0)=16#30000000  OR ADR(%MW0)=16#20000000 THEN (*841 or 881*)
						SysSockSetOption(
							diSocket:=m_Socket,
							diLevel:=6,
							diOption:=SOCKET_TCP_NODELAY,
							pOptionValue:=ADR(diOption),
							diOptionLength:=SIZEOF(diOption));
					ELSE
							;
					END_IF
					SysSockIoctl( m_Socket, SOCKET_FIONBIO, ADR(m_NoneBlocking));
					m_State:= STATE_RX;
					diError:=0;
				END_IF

		STATE_RX:
					m_BytesReceived:= SysSockRecv( m_Socket, ADR(m_ReceiveBuffer), SIZEOF(m_ReceiveBuffer), 0);
					CASE m_BytesReceived OF
					-1:(*no data available or error occured*)
						m_ConnectionWatchdog(IN:=TRUE , PT:=tServerTimeOut );
						IF m_connectionWatchdog.Q THEN
							m_State:= STATE_CLOSE;
							m_ConnectionWatchdog(IN:=FALSE);(*reset connection watchdog*)
							diError := 16#8009;
						END_IF
					0:(* socket was "gracefully closed"  *)
						m_State:= STATE_CLOSE;
						diError := 16#8003;
					ELSE
						(* Copy received data into receive buffer *)
						(********************************)
						FOR i:= 0 TO DINT_TO_INT(m_BytesReceived	)-1 DO
							aReceiveBuffer[diReceiveCount]:= m_ReceiveBuffer[i];
							diReceiveCount:=(diReceiveCount+1) MOD SIZEOF(aReceiveBuffer);
						END_FOR

						m_ConnectionWatchdog(IN:=FALSE);(*reset connection watchdog*)
					END_CASE

				(*send data*)
				IF xStartSend	 THEN
					m_State := STATE_TX;
				END_IF

	STATE_TX:	 (* send TCP-message *)
		m_diReturn := SysSockSend(diSocket := m_Socket,
								  pbyBuffer := ADR(ptSendData^[m_count]),(*geändert V1.4 bisher: [0] *)
								  diBufferSize := diSendCount-m_count,
								  diFlags :=m_Flags);
		CASE m_diReturn OF
		-1:	(* ERROR or data could not yet be send (V1.3 due to new FW11) *)
			m_ConnectionWatchdog(IN:=TRUE , PT:=tServerTimeOut );
			IF m_connectionWatchdog.Q THEN
				m_State:= STATE_CLOSE;
				m_ConnectionWatchdog(IN:=FALSE);(*reset connection watchdog*)
				diError := 16#8007;
			END_IF
		0: (* socket was "gracefully closed"  *)
			m_State := STATE_CLOSE;
			diError := 16#8003;
		ELSE (* succesful *)
			m_count:=m_count+m_diReturn;
			IF m_count>=diSendCount THEN
				diError := 16#0000;
				m_State := STATE_RX;
				m_count:=0;
				xStartSend:=FALSE;
			END_IF
			m_ConnectionWatchdog(IN:=FALSE);(*reset connection watchdog*)
		END_CASE


		STATE_CLOSE:	(* Close the server *)

		IF ADR(%MW0)=16#30000000  OR ADR(%MW0)=16#20000000 THEN (*841 or 881*)
			;
		ELSE
			IF m_Socket>=0 THEN
				SysSockShutdown(m_Socket, 0);;(*870*)
			END_IF
		END_IF
		IF m_Socket>=0 THEN
			SysSockClose( m_Socket);
		END_IF
		xClientConnected:= FALSE;
		m_State:= STATE_OPEN; (* Try to open the server again *)
		m_ConnectionWatchdog(IN:=FALSE);(*reset connection watchdog*)

		STATE_ERROR_TRAP: (* Error Read/Write socket  *)
			m_State:= STATE_ERROR_TRAP;

	ELSE  (* Bad FSM code trap  *)
			m_State:= STATE_ERROR_TRAP;
			diError:= 16#8008;
	END_CASE;
ELSE
	IF m_State <> STATE_INIT THEN
		IF ADR(%MW0)=16#30000000  OR ADR(%MW0)=16#20000000 THEN (*841 or 881*)
			;
		ELSE
			IF m_Socket>=0 THEN
				SysSockShutdown(m_Socket, 0);;(*870*)
			END_IF
		END_IF
		IF m_Socket>=0 THEN
			SysSockClose( m_Socket);
		END_IF
		IF ADR(%MW0)=16#30000000  OR ADR(%MW0)=16#20000000 THEN (*841 or 881*)
			;
		ELSE
			IF m_ServerSocket>=0 THEN
				SysSockShutdown(m_ServerSocket, 0);;(*870*)
			END_IF
		END_IF
		IF m_ServerSocket>=0 THEN
			SysSockClose( m_ServerSocket);
		END_IF
		xClientConnected:= FALSE;
		diError:= 0;
		m_State:= STATE_init; (* Try to open the server again *)
		m_ConnectionWatchdog(IN:=FALSE);(*reset connection watchdog*)
	END_IF
END_IF
END_FUNCTION_BLOCK

(* POU TCP_Logger/LogEv, ST *)
FUNCTION LogEv : BOOL
VAR_INPUT
	Level	: en_Logger_ErrLev;
	Object  : en_SYS_Objects;
	Index	: WORD;
	Error	: WORD;
	Message : STRING;
END_VAR
VAR
	s1 : STRING(160);
	i  : INT;
END_VAR
(* Execute error level operations *)
CASE Level OF
	EL_Wrn: 		Sys.Warning:=TRUE;
	EL_Alarm: 		Sys.Alarm:=TRUE;
	EL_AlarmStop: 	Sys.Alarm:=TRUE; (* GO TO STOP STATE!! *)
END_CASE

(* Fill lastlog list *)
s1:=CONCAT(Sys.Time_LogString,';Lev=');
s1:=CONCAT(s1,INT_TO_STRING(Level));
s1:=CONCAT(s1,';Obj=');
s1:=CONCAT(s1,INT_TO_STRING(Object));
s1:=CONCAT(s1,';Idx=');
s1:=CONCAT(s1,WORD_TO_STRING(Index));
s1:=CONCAT(s1,';Err=');
s1:=CONCAT(s1,WORD_TO_STRING(Error));
Sys.LastLogs_Dat[Sys.LastLogs_Idx]:=s1;
Sys.LastLogs_Msg[Sys.LastLogs_Idx]:=Message;
Sys.LastLogs_Idx:=Sys.LastLogs_Idx+1;
IF Sys.LastLogs_Idx>5 THEN Sys.LastLogs_Idx:=0; END_IF

(*---------------------------------------------------------------*)
(*---------------------------------------------------------------*)
Logger.TLen:=0;
(* Set GET header *)
ADDSTRING(ADR(Logger.TData), ADR(Logger_GETSTART), Logger.TLen);

(* Insert Header *)
s1:=INSERT('ID=&V=1&D=',DWORD_TO_STRING(Plant_SN),3);
s1:=CONCAT(s1,Sys.Time_LogString);
s1:=CONCAT(s1,'&S=');
IF Sys.Alarm THEN i:=2; ELSIF Sys.Warning THEN i:=1; ELSE i:=0; END_IF
s1:=CONCAT(s1,INT_TO_STRING(i));
ADDSTRING(ADR(Logger.TData), ADR(s1), Logger.TLen);

(* Insert ERR *)
s1:=CONCAT('&ERR=',INT_TO_STRING(Level));
s1:=CONCAT(s1,';');
s1:=CONCAT(s1,INT_TO_STRING(Object));
s1:=CONCAT(s1,';');
s1:=CONCAT(s1,WORD_TO_STRING(Index));
s1:=CONCAT(s1,';');
s1:=CONCAT(s1,WORD_TO_STRING(Error));
s1:=CONCAT(s1,';');
ADDSTRING(ADR(Logger.TData), ADR(s1), Logger.TLen);
s1:=Message;
STR_NOSPACES(ADR(s1));
ADDSTRING(ADR(Logger.TData), ADR(s1), Logger.TLen);

(* Finalize string *)
ADDSTRING(ADR(Logger.TData), ADR(Logger_GETEND), Logger.TLen);

(*---------------------------------------------------------------*)
(*---------------------------------------------------------------*)

Logger_Send();
END_FUNCTION

(* POU Utils Functions/ADDSTRING, ST *)
FUNCTION ADDSTRING : BOOL (* Append string to a byte buffer *)
VAR_INPUT
	pTxData: POINTER TO BYTE;
	pString: POINTER TO BYTE;
END_VAR
VAR_IN_OUT
	TxLen: DINT;
END_VAR
VAR
END_VAR
pTxData:=pTxData+TxLen;
WHILE pString^<>0 DO
	pTxData^:=pString^;
	pString:=pString+1;
	pTxData:=pTxData+1;
	TxLen:=TxLen+1;
END_WHILE
END_FUNCTION

(* POU Utils Functions/STR_NOSPACES, ST *)
FUNCTION STR_NOSPACES : BOOL (* Replace spaces and bad chars with allowed ones, used as HTTP-GET validator *)
VAR_INPUT
	pString: POINTER TO BYTE;
END_VAR
VAR
END_VAR
WHILE pString^<>0 DO
	IF pString^=16#20 (* space *) THEN pString^:=16#5F; (*'_'*) END_IF
	pString:=pString+1;
END_WHILE
END_FUNCTION

(* POU TCP_Logger/Logger_Send, ST *)
FUNCTION Logger_Send : BOOL
VAR
	hFile: 	DWORD;
	pos:	DWORD;
END_VAR
(* Read log position *)
pos:=SysFileGetSize(Logger_DataFile);
(* Check log size, bckup and erase if no pending messages *)
IF pos>100000000 (*100M*) THEN
	hFile:=SysFileOpen(Logger_IndexFile,'r');
	IF hFile=0 THEN
		SysFileDelete(Logger_DataFileOld);
		SysFileRename(Logger_DataFile,Logger_DataFileOld);
		pos:=0;
	ELSE
		SysFileClose(hFile);
	END_IF
END_IF
(* Write message on log file *)
hFile:=SysFileOpen(Logger_DataFile,'a');
IF hFile<>0 THEN
	SysFileWrite(hFile, ADR(Logger.TData), Logger.TLen);
	SysFileClose(hFile);
ELSE
	Sys.Warning:=TRUE;
END_IF


(* Check logger status *)
IF Logger.SendReq=FALSE THEN
	(* Set log position for recovery *)
	Logger.SendIdx:=pos;
	(* Copy message data *)
	MEMCPY(ADR(Logger.TData),ADR(Logger.SendData),DINT_TO_WORD(Logger.TLen));
	Logger.SendLen:=Logger.TLen;
	(* Trigger request *)
	Logger.SendReq:=TRUE;
ELSE
	(* Add message position+size in recovery indexes *)
	hFile:=SysFileOpen(Logger_IndexFile,'a');
	SysFileWrite(hFile, ADR(pos), SIZEOF(pos));
	SysFileWrite(hFile, ADR(Logger.TLen), SIZEOF(Logger.TLen));
	SysFileClose(hFile);
END_IF
END_FUNCTION

(* POU Utils Functions/MEMCPY, ST *)
FUNCTION MEMCPY:BOOL
VAR_INPUT
	pSourceAddress:POINTER TO ARRAY[1..2] OF BYTE;
	pDestinationAddress:POINTER TO ARRAY[1..2] OF BYTE;
	BytesToCopy:WORD;
END_VAR
VAR
END_VAR
WHILE (BytesToCopy > 0) DO
	pDestinationAddress^[1]:=pSourceAddress^[1]; (* copy bytes from source to destination *)
	pDestinationAddress:=ADR(pDestinationAddress^[2]); (* increment destination *)
	pSourceAddress:=ADR(pSourceAddress^[2]);(* increment source *)
	BytesToCopy:=BytesToCopy -1; (* decrement number of bytes to copy *)
END_WHILE
END_FUNCTION

(* POU Utils Functions/HEXTORAW, ST *)
FUNCTION HEXTORAW : WORD
VAR_INPUT
	pString		: POINTER TO BYTE;
	StringLen	: WORD;
	pData		: POINTER TO BYTE;
END_VAR
VAR
	xl: WORD;
	xi: WORD;
	xr: BYTE;
END_VAR
xl:=0;
xi:=0;

WHILE xi<StringLen DO

	IF pString^>=97 AND pString^<=102 THEN
		xr := pString^ - 87;
	ELSIF pString^>=65 AND pString^<=70 THEN
		xr := pString^ - 55;
	ELSIF pString^>=48 AND pString^<=57 THEN
		xr := pString^ - 48;
	ELSE
		xr := 16;
	END_IF

	IF xr<16 THEN
		IF (xi AND 1)=0 THEN
			pData^ := xr * 16;
		ELSE
			pData^ := pData^ + xr;
			pData := pData + 1;
			xl := xl + 1;
		END_IF
	END_IF

	xi := xi + 1;
	pString := pString + 1;

END_WHILE

HEXTORAW:=xl;
END_FUNCTION

(* POU Utils Functions/RAWTOHEX, ST *)
FUNCTION RAWTOHEX : WORD
VAR_INPUT
	pData: POINTER TO BYTE;
	DataLen: WORD;
	pString: POINTER TO BYTE;
END_VAR
VAR
	xl: WORD;
END_VAR
xl:=0;

WHILE DataLen>0 DO

	pString^ := (pData^ / 16#10) + 48 + (((pData^ / 16#10)/10)*7);
	pString:=pString+1;
	pString^ := (pData^ AND 16#0F)  + 48 + (((pData^ AND 16#0F)/10)*7);
	pString:=pString+1;
	pData:=pData+1;
	DataLen:=DataLen-1;
	xl:=xl+2;

END_WHILE

(*pString^:=0;*)

RAWTOHEX:=xl;
END_FUNCTION

(* POU Utils Functions/SetDataTime, ST *)
FUNCTION SetDataTime : DT
VAR_INPUT
	year : INT;
	month : INT;
	day : INT;
	hour : INT;
	minute : INT;
	second : INT;
END_VAR

VAR
	count : INT;
END_VAR
(* Creazione variabiletipo DT per creare Orario da dare al PLC *)


IF month > 2 THEN
	count := (month - 1) * 30;
	IF month > 7 THEN count := count + SHR(month - 3,1); ELSE count := count + SHR(month - 4,1); END_IF;
	(* chech for leap year and add one day if true *)
	IF SHL(year,14) = 0 THEN count := count + 1; END_IF;
ELSE
	count := (month - 1) * 31;
END_IF;


SetDataTime := DWORD_TO_DT(DATE_TO_DWORD( DWORD_TO_DATE((INT_TO_DWORD(count + day - 1) + SHR(INT_TO_DWORD(year) * 1461 - 2878169, 2)) * 86400))
				+ INT_TO_DWORD(SECOND)
				+ INT_TO_DWORD(MINUTE) * 60
				+ INT_TO_DWORD(HOUR) * 3600);
END_FUNCTION

(* POU Utils/USRLED_Update, ST *)
PROGRAM USRLED_Update
VAR
	OldStatus: en_SYS_Status;

	aFS : ARRAY [0..24] OF FLASHING_SEQUENCE :=
		(Colour:=GREEN,  Frequency:=1,   Relation:=128, Duration:=t#0s,    NextIndex:=0),  (* 0 => RUNNING *)
		(Colour:=ORANGE, Frequency:=1,   Relation:=128, Duration:=t#0s,    NextIndex:=1),  (* 1 => INIT *)
		(Colour:=RED,    Frequency:=4,   Relation:=128, Duration:=t#0s,    NextIndex:=2),  (* 2 => ERROR *)
		(Colour:=RED,    Frequency:=10,  Relation:=128, Duration:=t#0s,    NextIndex:=3),  (* 3 => ALARM *)
		(Colour:=ORANGE, Frequency:=200, Relation:=16,  Duration:=t#100ms, NextIndex:=11), (* 10 *)
		(Colour:=ORANGE, Frequency:=200, Relation:=32,  Duration:=t#100ms, NextIndex:=12),
		(Colour:=ORANGE, Frequency:=200, Relation:=64,  Duration:=t#100ms, NextIndex:=13),
		(Colour:=ORANGE, Frequency:=200, Relation:=128, Duration:=t#100ms, NextIndex:=14),
		(Colour:=ORANGE, Frequency:=200, Relation:=192, Duration:=t#100ms, NextIndex:=15),
		(Colour:=ORANGE, Frequency:=200, Relation:=128, Duration:=t#100ms, NextIndex:=16),
		(Colour:=ORANGE, Frequency:=200, Relation:=64,  Duration:=t#100ms, NextIndex:=17),
		(Colour:=ORANGE, Frequency:=200, Relation:=32,  Duration:=t#100ms, NextIndex:=18),
		(Colour:=ORANGE, Frequency:=200, Relation:=16,  Duration:=t#100ms, NextIndex:=19),
		(Colour:=ORANGE, Frequency:=200, Relation:=8,   Duration:=t#100ms, NextIndex:=10),
		(Colour:=GREEN,  Frequency:=200, Relation:=16,  Duration:=t#100ms, NextIndex:=21), (* 20 *)
		(Colour:=GREEN,  Frequency:=200, Relation:=32,  Duration:=t#100ms, NextIndex:=22),
		(Colour:=GREEN,  Frequency:=200, Relation:=64,  Duration:=t#100ms, NextIndex:=23),
		(Colour:=GREEN,  Frequency:=200, Relation:=128, Duration:=t#100ms, NextIndex:=24),
		(Colour:=GREEN,  Frequency:=200, Relation:=192, Duration:=t#100ms, NextIndex:=25),
		(Colour:=GREEN,  Frequency:=200, Relation:=128, Duration:=t#100ms, NextIndex:=26),
		(Colour:=GREEN,  Frequency:=200, Relation:=64,  Duration:=t#100ms, NextIndex:=27),
		(Colour:=GREEN,  Frequency:=200, Relation:=32,  Duration:=t#100ms, NextIndex:=28),
		(Colour:=GREEN,  Frequency:=200, Relation:=16,  Duration:=t#100ms, NextIndex:=29),
		(Colour:=GREEN,  Frequency:=200, Relation:=8,   Duration:=t#100ms, NextIndex:=20);

	pFS : POINTER TO FLASHING_SEQUENCE;


END_VAR
IF Sys.Status <> OldStatus THEN

	OldStatus:=Sys.Status;

	CASE OldStatus OF

		S_STARTUP:
			pFS:=ADR(aFS);
			SET_FLASHING_SEQUENCE(EN:=TRUE, POINTER_TO_POINTER_TO_ARRAY:=ADR(pFS));
			SET_FLASHING_SEQUENCE_INDEX(EN:=TRUE, IMMEDIATE:=FALSE, INDEX:=1);
			START_FLASHING_SEQUENCE(EN:=TRUE);

		S_RUNNING:
			SET_FLASHING_SEQUENCE_INDEX(EN:=TRUE, IMMEDIATE:=TRUE, INDEX:=0);

	END_CASE

END_IF
END_PROGRAM

(* POU Plant/SYS_Proc, ST *)
PROGRAM SYS_Proc
VAR
(*	fALARM_PB		:FLT_TAP;
	fALARM_TB		:FLT_TAP;
	fALARM_PM		:FLT_TAP; *)

(*	fGZB_ST			:FLT_TAP; (* GATEWAY ZIGBEE *)*)
(*	fVPN_OUT1		:FLT_TAP; (* VPN - CONNECT *)*)
	fVPN_OUT2		:FLT_TAP; (* VPN - STATUS *)
(*	fKEY_CT_ST		:FLT_TAP; (* DOOR01 - Porta primaria *)*)
(*	fKEY_SCT_ST		:FLT_TAP; (* DOOR02 - Porta secondaria *)*)
	fKEY_QE_ST		:FLT_TAP; (* DOOR03 - Quadro Elettrico *)

END_VAR
(*************** ISPESL *****************)
(*
fALARM_PB(IN:=ALARM_PB);
IF fALARM_PB.EVH THEN
	LogEv(EL_AlarmStop,EO_PBV,1,1,'Over_Pressure_Alarm');
END_IF

fALARM_TB(IN:=ALARM_TB);
IF fALARM_TB.EVH THEN
	LogEv(EL_AlarmStop,EO_TBV,1,1,'Over_Temperature_Alarm');
END_IF

fALARM_PM(IN:=ALARM_PM);
IF fALARM_PM.EVH THEN
	LogEv(EL_AlarmStop,EO_PMV,1,1,'Under_Pressure_Alarm');
END_IF
*)
(****************************************)

(*### VPN Connection Check ###*)(*
fVPN_OUT1(IN:=VPN_OUT1);
IF fVPN_OUT1.EVH THEN
	LogEv(EL_Log,EO_VPN,1,1,'CONNECT_ON');
END_IF
IF fVPN_OUT1.EVL THEN
	LogEv(EL_Log,EO_VPN,1,2,'CONNECT_OFF');
END_IF*)

(*### VPN Status Check ###*)
fVPN_OUT2(IN:=VPN_OUT2);
IF fVPN_OUT2.EVH THEN
	LogEv(EL_Log,EO_VPN,1,3,'STATUS_UP');
END_IF
IF fVPN_OUT2.EVL THEN
	LogEv(EL_Wrn,EO_VPN,1,4,'STATUS_DOWN');
END_IF

(*### DOOR01 Status Check ###*)(*
fKEY_CT_ST(IN:=KEY_CT_ST);
IF fKEY_CT_ST.EVH THEN
	LogEv(EL_Log,EO_DOOR,1,2,'Centrale_termica_Close');
END_IF
IF fKEY_CT_ST.EVL THEN
	LogEv(EL_Wrn,EO_DOOR,1,1,'Centrale_termica_Open');
END_IF*)

(*### DOOR02 Status Check ###*)(*
fKEY_SCT_ST(IN:=KEY_SCT_ST);
IF fKEY_SCT_ST.EVH THEN
	LogEv(EL_Log,EO_DOOR,2,2,'Sottocentrale_termica_Close');
END_IF
IF fKEY_SCT_ST.EVL THEN
	LogEv(EL_Wrn,EO_DOOR,2,1,'Sottocentrale_termica_Open');
END_IF*)

(*### DOOR03 Status Check ###*)
fKEY_QE_ST(IN:=KEY_QE_ST);
IF fKEY_QE_ST.EVH THEN
	LogEv(EL_Log,EO_DOOR,3,2,'Quadro_Close');
END_IF
IF fKEY_QE_ST.EVL THEN
	LogEv(EL_Wrn,EO_DOOR,3,1,'Quadro_Open');
END_IF
END_PROGRAM

(* POU Utils Functions/FLT_TAP, ST *)
FUNCTION_BLOCK FLT_TAP
VAR_INPUT
	IN		: BOOL;
	TAP		: BYTE:=4;
	INITEV	: BOOL:=TRUE;
END_VAR
VAR_OUTPUT
	OUT		: BOOL;
	EVH		: BOOL;
	EVL		: BOOL;
END_VAR
VAR
	init	: BOOL:=FALSE;
	cnt		: BYTE;
END_VAR
EVH:=FALSE;
EVL:=FALSE;

IF NOT init THEN
	init := TRUE;
	IF INITEV THEN
		OUT  := NOT IN;
		cnt  := TAP;
	ELSE
		OUT  := IN;
	END_IF
END_IF

IF OUT<>IN THEN
	cnt:=cnt+1;
	IF cnt>TAP THEN
		OUT:=IN;
		cnt:=0;
		IF OUT THEN EVH:=TRUE; ELSE EVL:=TRUE; END_IF
	END_IF
ELSE
	cnt:=0;
END_IF
END_FUNCTION_BLOCK

(* POU Utils Functions/AVERAGE_T, ST *)
FUNCTION_BLOCK AVERAGE_T
VAR_INPUT
	IN: 	INT;
END_VAR
VAR_OUTPUT
	HI:		INT;
	AVG:	INT;
	LOW:	INT;
	ERR:	BOOL;
END_VAR
VAR
	sum:	DINT;
	cnt:	WORD;
END_VAR
IF cnt>=65000 THEN
	ERR:=TRUE;
	Read();
	sum := sum - AVG;
	cnt := cnt + 1;
END_IF

sum := sum + IN;
cnt := cnt + 1;

IF IN<LOW THEN  LOW:=IN; END_IF
IF IN>HI  THEN HI :=IN; END_IF
END_FUNCTION_BLOCK
ACTION Read:
AVG := DINT_TO_INT(sum/cnt);
END_ACTION
ACTION Reset:
HI:=IN;
AVG:=IN;
LOW:=IN;
ERR:=FALSE;

sum:=IN;
cnt:=1;
END_ACTION

(* POU Utils Functions/COPY_32SWAP16, ST *)
FUNCTION COPY_32SWAP16:BOOL
VAR_INPUT
	pSourceAddress		:POINTER TO ARRAY[1..2] OF WORD;
	pDestinationAddress	:POINTER TO ARRAY[1..2] OF WORD;
END_VAR
VAR
END_VAR
pDestinationAddress^[1]:=pSourceAddress^[2];
pDestinationAddress^[2]:=pSourceAddress^[1];
END_FUNCTION

(* POU Utils Functions/FLT_EVENT, ST *)
FUNCTION_BLOCK FLT_EVENT
VAR_INPUT
	IN		: BOOL;
	INITEV	: BOOL:=TRUE;
END_VAR
VAR_OUTPUT
	EVH		: BOOL;
	EVL		: BOOL;
END_VAR
VAR
	init	: BOOL:=FALSE;
	old		: BOOL;
END_VAR
EVH:=FALSE;
EVL:=FALSE;

IF NOT init THEN
	init:=TRUE;
	IF INITEV THEN
		old := NOT IN;
	ELSE
		old := IN;
	END_IF
END_IF

IF old<>IN THEN
	old:=IN;
	IF IN THEN EVH:=TRUE; ELSE EVL:=TRUE; END_IF
END_IF
END_FUNCTION_BLOCK

(* POU Utils Functions/FLT_TIME, ST *)
FUNCTION_BLOCK FLT_TIME
VAR_INPUT
	IN		: BOOL;
	TTAP	: TIME:=T#5s;
	INITEV	: BOOL:=TRUE;
END_VAR
VAR_OUTPUT
	OUT		: BOOL;
	EVH		: BOOL;
	EVL		: BOOL;
END_VAR
VAR
	init	: BOOL:=FALSE;
	timer	: TON;
END_VAR
EVH:=FALSE;
EVL:=FALSE;

IF NOT init THEN
	init := TRUE;
	IF INITEV THEN
		OUT  := NOT IN;
	ELSE
		OUT  := IN;
	END_IF
END_IF

IF OUT<>IN THEN
	timer(IN:=TRUE,PT:=TTAP);
	IF timer.Q THEN
		OUT:=IN;
		timer(IN:=FALSE);
		IF OUT THEN EVH:=TRUE; ELSE EVL:=TRUE; END_IF
	END_IF
ELSE
	timer(IN:=FALSE);
END_IF
END_FUNCTION_BLOCK

(* POU TCP_Logger/LogTrig, ST *)
FUNCTION LogTrig : BOOL
VAR
	s1 : STRING(160);
	i  : BYTE;
	j  : WORD;
END_VAR
(*---------------------------------------------------------------*)
(*---------------------------------------------------------------*)
Logger.TLen:=0;
(* Set GET header *)
ADDSTRING(ADR(Logger.TData), ADR(Logger_GETSTART), Logger.TLen);

(* Insert Header *)
s1:=INSERT('ID=&V=1&D=',DWORD_TO_STRING(Plant_SN),3);
s1:=CONCAT(s1,Sys.Time_LogString);
s1:=CONCAT(s1,'&S=');
IF Sys.Alarm THEN i:=2; ELSIF Sys.Warning THEN i:=1; ELSE i:=0; END_IF
s1:=CONCAT(s1,BYTE_TO_STRING(i));
ADDSTRING(ADR(Logger.TData), ADR(s1), Logger.TLen);

(* Insert contabilizers  *)
GAS02.AddLogData( MODBUS:=MODB01 );
CTB05.AddLogData( MBUS:=MBUS01 );
CTB06.AddLogData( MBUS:=MBUS01 );
CTB07.AddLogData( MBUS:=MBUS01 );

(* Finalize string *)
ADDSTRING(ADR(Logger.TData), ADR(Logger_GETEND), Logger.TLen);

(*---------------------------------------------------------------*)
(*---------------------------------------------------------------*)

Logger_Send();
END_FUNCTION

(* POU Utils Functions/MEMCLR, ST *)
FUNCTION MEMCLR:BOOL
VAR_INPUT
	pDestinationAddress:POINTER TO ARRAY[1..2] OF BYTE;
	BytesToClear:WORD;
END_VAR
VAR
END_VAR
WHILE (BytesToClear > 0) DO
	pDestinationAddress^[1]:=0;
	pDestinationAddress:=ADR(pDestinationAddress^[2]); (* increment destination *)
	BytesToClear:=BytesToClear -1; (* decrement number of bytes to copy *)
END_WHILE
END_FUNCTION

(* POU Plant_Objects/obj_MBUS, ST *)
FUNCTION_BLOCK obj_MBUS
(* === M-BUS PROTOCOL INTERFACE ===
   v1.0[16/03/05] - Added interface errors
*)
VAR_INPUT
	(* Settings *)
	ID				: BYTE;
	COM				: BYTE;
	BAUDRATE		: COM_BAUDRATE;
	(* Interface *)
	MBus 			: typMBus;
	MBus_Master 	: FbMBusMaster;
END_VAR
VAR_OUTPUT
	(* Status *)
	Status_Log		: BYTE;
	Status_Vis 		: DWORD;
END_VAR
VAR
	Alarm			: FLT_EVENT;
END_VAR
MBus_Master( bCOMPORT:=COM , enumBAUDRATE:=BAUDRATE , utMBus:=MBus );

(* Check status *)
Alarm(IN:=(MBus.bCOM_ERROR<>0));
IF Alarm.EVH THEN
	LogEv(EL_Alarm,EO_MBUS,ID,1,BYTE_TO_STRING(MBus.bCOM_ERROR));
END_IF
IF Alarm.EVL THEN
	LogEv(EL_Log,EO_MBUS,ID,2,'MBUS_OK');
END_IF

(* Log/visu status *)
   IF Alarm.IN   					THEN Status_Log:=2; Status_Vis:=16#2020F0;
ELSIF (MBus.bL1_ERROR AND 16#1F)<>0 THEN Status_Log:=1; Status_Vis:=16#20F0F0;
  				 					ELSE Status_Log:=0; Status_Vis:=16#20F020;
END_IF
END_FUNCTION_BLOCK

(* POU Plant_Objects/obj_MBUS_CTB_SHARKY775, ST *)
FUNCTION_BLOCK obj_MBUS_CTB_SHARKY775
(* === M-BUS CONTABILIZER SHARKY 775 ===
   v1.0[16/03/05] - Error management
*)
VAR_INPUT
	(* Settings *)
	ID				: BYTE;
	ADDRESS			: DWORD;
	Refresh_Period	: TIME:=t#3m;
	(* Controls *)
	Refresh_Auto	: BOOL:=TRUE; (* Enable automatic refresh *)
	Refresh_Now		: BOOL; 	  (* Force an immediate refresh *)
END_VAR
VAR_IN_OUT
	(* Interface *)
	MBUS			: obj_MBUS;
END_VAR
VAR_OUTPUT
	M1				: FbMBus_Heat;
	(* Status *)
	Status_Log		: BYTE;
	Status_Vis 		: DWORD;
END_VAR
VAR
	dly 	 	: TON := (PT:=t#5s);
	M1_Start	: BOOL;

	init_st		: BOOL;
	bus_st0		: BYTE;
	dev_st0		: BYTE;

(*	S1			: FbMBusSend;
	S1_Start	: BOOL;*)
(*	C1			: FbUnitConverter; *)
END_VAR
(* Auto refresh timer *)
dly(IN:=NOT (dly.Q OR Refresh_Now OR (NOT Refresh_Auto)));
(* Trigger refresh *)
IF dly.Q OR Refresh_Now THEN
	dly.PT:=Refresh_Period;
	Refresh_Now:=FALSE;
	(* Start reading *)
	M1.dwAdr:= ADDRESS;
	M1.xSND_NKE:=TRUE;
	M1_Start:=TRUE;
END_IF

(* Contabilizer module *)
M1(	utMBus:=MBUS.MBus, xStart:=M1_Start );

(* Extra actions *)
(*C1( utMBus:=MBUS.MBus, xStart:=C1_Start );*)

(* Check status *)
IF NOT init_st OR M1.bError<>bus_st0 OR M1.utMBInfo.bMStatus<>dev_st0 THEN
	init_st:=TRUE;
	bus_st0:=M1.bError; dev_st0:=M1.utMBInfo.bMStatus;
	IF bus_st0<>0 THEN
		LogEv(EL_Alarm,EO_CTB,ID,2,BYTE_TO_STRING(bus_st0));
		Status_Log:=2; Status_Vis:=16#2020F0;
	ELSE
		IF dev_st0<>0 THEN
			Status_Log:=2; Status_Vis:=16#2020F0;
			CASE dev_st0 OF
				16#08: LogEv(EL_Alarm,EO_CTB,ID,10,'C-1');
				16#04: LogEv(EL_Alarm,EO_CTB,ID,10,'E-8');
				16#28: LogEv(EL_Alarm,EO_CTB,ID,10,'E-4');
				16#50: LogEv(EL_Alarm,EO_CTB,ID,10,'E-1');
				16#70: LogEv(EL_Alarm,EO_CTB,ID,10,'E-7');
				16#84: LogEv(EL_Alarm,EO_CTB,ID,10,'E-9');
				16#B0: LogEv(EL_Wrn  ,EO_CTB,ID,10,'E-3');
				16#D0: LogEv(EL_Wrn  ,EO_CTB,ID,10,'E-6');
				16#F0: LogEv(EL_Alarm,EO_CTB,ID,10,'Leak');
				16#10: LogEv(EL_Wrn  ,EO_CTB,ID,10,'E-5'); Status_Log:=1; Status_Vis:=16#20F0F0;
			ELSE
				LogEv(EL_Alarm,EO_CTB,ID,10,BYTE_TO_STRING(dev_st0));
			END_CASE
		ELSE
			Status_Log:=0; Status_Vis:=16#20F020;
			LogEv(EL_Log,EO_CTB,ID,1,'');
		END_IF
	END_IF
END_IF
END_FUNCTION_BLOCK
ACTION AddLogData:
Logger.s1:=INSERT('&CTB=',BYTE_TO_STRING(ID),4);
IF ID<10 THEN Logger.s1:=INSERT(Logger.s1,'0',4); END_IF

Logger.s1:=CONCAT(Logger.s1,M1.utFTemp.Value);		Logger.s1:=CONCAT(Logger.s1,';');
Logger.s1:=CONCAT(Logger.s1,M1.utRTemp.Value);		Logger.s1:=CONCAT(Logger.s1,';');
Logger.s1:=CONCAT(Logger.s1,M1.utFlow.Value);		Logger.s1:=CONCAT(Logger.s1,';');
Logger.s1:=CONCAT(Logger.s1,M1.utPower.Value);		Logger.s1:=CONCAT(Logger.s1,';');
Logger.s1:=CONCAT(Logger.s1,M1.utEnergy.Value);		Logger.s1:=CONCAT(Logger.s1,';');

Logger.s1:=CONCAT(Logger.s1,BYTE_TO_STRING(Status_Log));
ADDSTRING(ADR(Logger.TData), ADR(Logger.s1), Logger.TLen);
END_ACTION

(* POU Plant_Objects/obj_MODBUS, ST *)
FUNCTION_BLOCK obj_MODBUS
(* === MODBUS PROTOCOL INTERFACE ===
   v1.0[16/03/05] - Support for RS485 half-duplex
				  - Rewritten vars management with state machine
   v1.1[27/03/05] - Fixed vars manager & introduced retry before alarm
   v1.2[16/04/05] - Changed initialization alarm to a simple warning
   v1.3[20/04/05] - Var alarm auto-recover when succesful reading of last error variable
*)
VAR CONSTANT
	VARS_Max	: BYTE := 32;
END_VAR
VAR_INPUT
	(* Settings *)
	ID			: BYTE;
	COM			: BYTE;
	BAUDRATE	: COM_BAUDRATE;
	RS485		: BOOL := FALSE;
	(* Interface *)
	MB_MASTER	: MODBUS_EXTENDED_MASTER;
	MB_Start	: BOOL;
	MB_Query	: typModbusExtendedQuery;
	MB_Resp		: typModbusResponse;
	MB_Lock		: BOOL;
	(* Variables management *)
	VARS_En		: BOOL;
	VARS		: ARRAY [0..VARS_Max] OF typ_MODBUS_VAR;
	VARS_Check	: BOOL;
	VARS_Alarm	: BOOL;
END_VAR
VAR_OUTPUT
	(* Status *)
	Status_Log	: BYTE;
	Status_Vis	: DWORD;
END_VAR
VAR
	i			: BYTE;
	Alarm		: FLT_EVENT;
	VarTmr		: TON := (PT:=T#1s);
	VarSta		: BYTE; (* Status *)
	VarCnt		: BYTE; (* Scan counter *)
	VarRetry	: BYTE;
	VarAlarm	: BYTE; (* Last variable with errors *)
END_VAR
MB_MASTER(
	ENABLE:=TRUE ,
	ASCII_Mode:=FALSE,
	bCOM_PORT:=COM ,
	cbCOM_BAUDRATE:=BAUDRATE ,
	cpCOM_PARITY:=PARITY_NO ,
	csCOM_STOPBITS:=STOPBITS_1 ,
	cbsCOM_BYTESIZE:=BS_8 ,
	cfCOM_FLOW_CONTROL:=SEL(RS485,NO_FLOW_CONTROL,HALFDUPLEX) ,
	tTIME_OUT:=t#250ms ,
	StartFunction:=MB_Start ,
	ExtQuery:=MB_Query ,
	Response:=MB_Resp  );

(* Process variable management *)
IF VARS_En THEN VARS_Process(); END_IF

(* Check status *)
Alarm(IN:=(MB_MASTER.bInterfaceError<>0));
IF Alarm.EVH THEN
	LogEv(SEL(MB_MASTER.bInterfaceError<>3,EL_Wrn,EL_Alarm),EO_MODBUS,ID,1,BYTE_TO_STRING(MB_MASTER.bInterfaceError));
END_IF
IF Alarm.EVL THEN
	LogEv(EL_Log,EO_MODBUS,ID,2,'MODBUS_OK');
END_IF

(* Log/visu status *)
   IF Alarm.IN   THEN Status_Log:=2; Status_Vis:=16#2020F0;
ELSIF Vars_Alarm THEN Status_Log:=1; Status_Vis:=16#20F0F0;
  				 ELSE Status_Log:=0; Status_Vis:=16#20F020;
END_IF
END_FUNCTION_BLOCK
ACTION VARS_Process:
(* Update var timers *)
VarTmr(IN:=(NOT VarTmr.Q));
IF VarTmr.Q THEN
	FOR i := 0 TO VARS_Max DO
		IF VARS[i].Refresh_Cnt>0 THEN VARS[i].Refresh_Cnt:=VARS[i].Refresh_Cnt-1; END_IF
	END_FOR
	VARS_Check:=TRUE;
END_IF


(* Process status *)
CASE VarSta OF
	0: (* === Init *)
		VarCnt:=0;
		VarSta:=1;

	1: (* === Wait check signal *)
		IF VARS_Check THEN
			VARS_Check:=FALSE;
			VarCnt:=0;
			VarSta:=2;
		END_IF

	2: (* === Check loop *)
		IF NOT (MB_Lock OR MB_Start) THEN
			WHILE VarCnt<=VARS_Max AND VarSta=2 DO
				(* Check only active vars *)
				IF VARS[VarCnt].SlaveAddress<>0 THEN
					(* Check var auto-refresh on timer checks *)
					IF VARS[VarCnt].Refresh_Time>0 AND VARS[VarCnt].Refresh_Cnt=0 THEN
						VARS[VarCnt].Refresh_Cnt:=VARS[VarCnt].Refresh_Time;
						VarSta:=3;
					END_IF
					(* Check refresh for change or request *)
					CASE VARS[VarCnt].FunCode OF
						16#5,16#6,16#F,16#10:
							IF VARS[VarCnt].Variable^<>VARS[VarCnt].Variable_Mirror THEN
								VARS[VarCnt].Variable_Mirror:=VARS[VarCnt].Variable^;
								VarSta:=3;
							END_IF
						16#1,16#2,16#3,16#4:
							IF VARS[VarCnt].Variable_Mirror<>0 THEN
								VARS[VarCnt].Variable_Mirror:=0;
								VarSta:=3;
							END_IF
					END_CASE
				END_IF
				(* Process query *)
				IF VarSta=3 THEN
					MB_Lock:=TRUE;
					MB_Query.SlaveAddress:=VARS[VarCnt].SlaveAddress;
					MB_Query.FunctionCode:=VARS[VarCnt].FunCode;
					CASE VARS[VarCnt].FunCode OF
						16#5,16#6,16#F,16#10:
							MB_Query.Read_StartAddress:=0;
							MB_Query.Read_Quantity:=0;
							MB_Query.Write_StartAddress:=VARS[VarCnt].FunAddress;
							MB_Query.Write_Quantity:=VARS[VarCnt].Variable_Size;
							MB_Query.Write_Data[0]:=VARS[VarCnt].Variable^;
						16#1,16#2,16#3,16#4:
							MB_Query.Read_StartAddress:=VARS[VarCnt].FunAddress;
							IF VARS[VarCnt].Variable_Size=200 THEN MB_Query.Read_Quantity:=2; ELSE
							  MB_Query.Read_Quantity:=VARS[VarCnt].Variable_Size;
							END_IF
							MB_Query.Write_StartAddress:=0;
							MB_Query.Write_Quantity:=0;
					END_CASE
					VarRetry:=0;
					MB_Start:=TRUE;
				ELSE
					VarCnt:=VarCnt+1;
				END_IF
			END_WHILE
			(* Check loop completed -> no actions *)
			IF VarSta=2 THEN VarSta:=1; END_IF
		END_IF

	3: (* === Wait & process MB response *)
		IF NOT MB_Start THEN
			IF MB_MASTER.MB_Error=0 THEN
				CASE VARS[VarCnt].FunCode OF
					16#1,16#2,16#3,16#4:
						IF VARS[VarCnt].Variable_Size=200 THEN
							COPY_32SWAP16(ADR(MB_Resp.Data), VARS[VarCnt].Variable);
						ELSIF VARS[VarCnt].Variable_Size>1 THEN
							MEMCPY(ADR(MB_Resp.Data), VARS[VarCnt].Variable, 2*VARS[VarCnt].Variable_Size);
						ELSE
							VARS[VarCnt].Variable^:=MB_Resp.Data[0];
						END_IF
				END_CASE
				MB_Lock:=FALSE;
				(* Signal error recovery *)
				IF VARS_Alarm=TRUE AND VarCnt=VarAlarm THEN
					LogEv(EL_Wrn,EO_MODBUS,ID,5,'');
					VARS_Alarm:=FALSE;
				END_IF
				(* Next var *)
				VarCnt:=VarCnt+1;
				VarSta:=2;
			ELSE
				IF VarRetry<3 THEN
					VarRetry:=VarRetry+1;
					MB_Start:=TRUE;
				ELSE
					MB_Lock:=FALSE;
					(* Signal error *)
					IF VARS_Alarm=FALSE THEN
						LogEv(EL_Wrn,EO_MODBUS,ID,3,INT_TO_STRING(MB_MASTER.MB_Error));
						VARS_Alarm:=TRUE;
						VarAlarm:=VarCnt-1;
					END_IF
					(* Next var *)
					VarCnt:=VarCnt+1;
					VarSta:=2;
				END_IF
			END_IF
		END_IF

ELSE
	VarSta:=0;
END_CASE
END_ACTION

(* POU Plant_Objects/obj_MODBUS_ELGAS_MINIELCOR, ST *)
FUNCTION_BLOCK obj_MODBUS_ELGAS_MINIELCOR
VAR_INPUT
	(* Settings *)
	ID				: BYTE;
	ADDRESS			: BYTE:=1;
(*	Refresh_Period	: TIME:=t#1m30s;*)
	Refresh_Time	: BYTE:=180;
	(* Controls *)
(*	Refresh_Auto	: BOOL; (* Enable automatic refresh *)*)
(*	Refresh_Now		: BOOL; (* Force an immediate refresh *)*)
END_VAR
VAR_IN_OUT
	MODBUS			: obj_MODBUS;
END_VAR
VAR_OUTPUT
	Data			: typ_MODBUS_ELGAS_MINIELCOR;
	(* Status *)
	Status_Log		: BYTE;
	Status_Vis 		: DWORD;
END_VAR
VAR
	sta		: BYTE; 	(* Status *)
	Alarm	: FLT_EVENT;

(*	dly 	: TON := (PT:=t#5s);
	addr 	: WORD:=19;
	siz		: WORD:=2;*)

END_VAR
CASE sta OF

	0: (* === Initialize *)

		MODBUS.VARS[0].SlaveAddress:=1;
		MODBUS.VARS[0].FunCode:=3;
		MODBUS.VARS[0].FunAddress:=3;
		MODBUS.VARS[0].Refresh_Time:=Refresh_Time;
		MODBUS.VARS[0].Variable_Mirror:=0;
		MODBUS.VARS[0].Variable_Size:=4;
		MODBUS.VARS[0].Variable:=ADR(Data.Vb);

		MODBUS.VARS[1].SlaveAddress:=1;
		MODBUS.VARS[1].FunCode:=3;
		MODBUS.VARS[1].FunAddress:=19;
		MODBUS.VARS[1].Refresh_Time:=Refresh_Time;
		MODBUS.VARS[1].Variable_Mirror:=0;
		MODBUS.VARS[1].Variable_Size:=200;
		MODBUS.VARS[1].Variable:=ADR(Data.Vm);

		MODBUS.VARS[2].SlaveAddress:=1;
		MODBUS.VARS[2].FunCode:=3;
		MODBUS.VARS[2].FunAddress:=25;
		MODBUS.VARS[2].Refresh_Time:=Refresh_Time;
		MODBUS.VARS[2].Variable_Mirror:=0;
		MODBUS.VARS[2].Variable_Size:=200;
		MODBUS.VARS[2].Variable:=ADR(Data.P);

		MODBUS.VARS[3].SlaveAddress:=1;
		MODBUS.VARS[3].FunCode:=3;
		MODBUS.VARS[3].FunAddress:=27;
		MODBUS.VARS[3].Refresh_Time:=Refresh_Time;
		MODBUS.VARS[3].Variable_Mirror:=0;
		MODBUS.VARS[3].Variable_Size:=200;
		MODBUS.VARS[3].Variable:=ADR(Data.T);

		MODBUS.VARS[4].SlaveAddress:=1;
		MODBUS.VARS[4].FunCode:=3;
		MODBUS.VARS[4].FunAddress:=39;
		MODBUS.VARS[4].Refresh_Time:=Refresh_Time;
		MODBUS.VARS[4].Variable_Mirror:=0;
		MODBUS.VARS[4].Variable_Size:=200;
		MODBUS.VARS[4].Variable:=ADR(Data.C);

		MODBUS.VARS[5].SlaveAddress:=1;
		MODBUS.VARS[5].FunCode:=3;
		MODBUS.VARS[5].FunAddress:=7;
		MODBUS.VARS[5].Refresh_Time:=Refresh_Time;
		MODBUS.VARS[5].Variable_Mirror:=0;
		MODBUS.VARS[5].Variable_Size:=4;
		MODBUS.VARS[5].Variable:=ADR(Data.Vbs);

		MODBUS.VARS[6].SlaveAddress:=1;
		MODBUS.VARS[6].FunCode:=3;
		MODBUS.VARS[6].FunAddress:=11;
		MODBUS.VARS[6].Refresh_Time:=Refresh_Time;
		MODBUS.VARS[6].Variable_Mirror:=0;
		MODBUS.VARS[6].Variable_Size:=4;
		MODBUS.VARS[6].Variable:=ADR(Data.Vb_d_d);

		MODBUS.VARS[7].SlaveAddress:=1;
		MODBUS.VARS[7].FunCode:=3;
		MODBUS.VARS[7].FunAddress:=15;
		MODBUS.VARS[7].Refresh_Time:=Refresh_Time;
		MODBUS.VARS[7].Variable_Mirror:=0;
		MODBUS.VARS[7].Variable_Size:=4;
		MODBUS.VARS[7].Variable:=ADR(Data.Vb_d_m);

		MODBUS.VARS[8].SlaveAddress:=1;
		MODBUS.VARS[8].FunCode:=3;
		MODBUS.VARS[8].FunAddress:=21;
		MODBUS.VARS[8].Refresh_Time:=Refresh_Time;
		MODBUS.VARS[8].Variable_Mirror:=0;
		MODBUS.VARS[8].Variable_Size:=200;
		MODBUS.VARS[8].Variable:=ADR(Data.Vm_d_d);

		MODBUS.VARS[9].SlaveAddress:=1;
		MODBUS.VARS[9].FunCode:=3;
		MODBUS.VARS[9].FunAddress:=31;
		MODBUS.VARS[9].Refresh_Time:=Refresh_Time;
		MODBUS.VARS[9].Variable_Mirror:=0;
		MODBUS.VARS[9].Variable_Size:=200;
		MODBUS.VARS[9].Variable:=ADR(Data.BC_EVC);

		MODBUS.VARS[10].SlaveAddress:=1;
		MODBUS.VARS[10].FunCode:=3;
		MODBUS.VARS[10].FunAddress:=29;
		MODBUS.VARS[10].Refresh_Time:=Refresh_Time;
		MODBUS.VARS[10].Variable_Mirror:=0;
		MODBUS.VARS[10].Variable_Size:=200;
		MODBUS.VARS[10].Variable:=ADR(Data.BV_EVC);

		MODBUS.VARS[11].SlaveAddress:=1;
		MODBUS.VARS[11].FunCode:=3;
		MODBUS.VARS[11].FunAddress:=35;
		MODBUS.VARS[11].Refresh_Time:=Refresh_Time;
		MODBUS.VARS[11].Variable_Mirror:=0;
		MODBUS.VARS[11].Variable_Size:=200;
		MODBUS.VARS[11].Variable:=ADR(Data.Q);

		MODBUS.VARS[12].SlaveAddress:=1;
		MODBUS.VARS[12].FunCode:=3;
		MODBUS.VARS[12].FunAddress:=37;
		MODBUS.VARS[12].Refresh_Time:=Refresh_Time;
		MODBUS.VARS[12].Variable_Mirror:=0;
		MODBUS.VARS[12].Variable_Size:=200;
		MODBUS.VARS[12].Variable:=ADR(Data.Qb);

		MODBUS.VARS[13].SlaveAddress:=1;
		MODBUS.VARS[13].FunCode:=3;
		MODBUS.VARS[13].FunAddress:=55;
		MODBUS.VARS[13].Refresh_Time:=Refresh_Time;
		MODBUS.VARS[13].Variable_Mirror:=0;
		MODBUS.VARS[13].Variable_Size:=1;
		MODBUS.VARS[13].Variable:=ADR(Data.D_Err);

		MODBUS.VARS[14].SlaveAddress:=1;
		MODBUS.VARS[14].FunCode:=3;
		MODBUS.VARS[14].FunAddress:=56;
		MODBUS.VARS[14].Refresh_Time:=Refresh_Time;
		MODBUS.VARS[14].Variable_Mirror:=0;
		MODBUS.VARS[14].Variable_Size:=200;
		MODBUS.VARS[14].Variable:=ADR(Data.Status);

		MODBUS.VARS_En:=TRUE;

		sta:=1;

	1:	(* === Check status *)
		Alarm(IN:=(Data.D_Err<>0));
		IF Alarm.EVL THEN
			LogEv(EL_Log,EO_GAS,ID,1,'');
		END_IF
		IF Alarm.EVH THEN
			LogEv(EL_Alarm,EO_GAS,ID,3,DWORD_TO_STRING(Data.Status));
		END_IF

		(* Log/visu status *)
		   IF Alarm.IN   		THEN Status_Log:=2; Status_Vis:=16#2020F0;
		ELSIF MODBUS.Vars_Alarm THEN Status_Log:=1; Status_Vis:=16#20F0F0;
		  				 		ELSE Status_Log:=0; Status_Vis:=16#20F020;
		END_IF

(*
	1: (* === Wait update signals *)
		dly(IN:=NOT (dly.Q OR Refresh_Now OR (NOT Refresh_Auto)));
		IF dly.Q OR Refresh_Now THEN
			dly.PT:=Refresh_Period;
			Refresh_Now:=FALSE;
			sta:=2;
		END_IF

	2: (* === Start update when MB is free *)
		IF NOT (MODBUS.MB_Lock OR MODBUS.MB_Start) THEN
			MODBUS.MB_Lock:=TRUE;
			MODBUS.MB_Query.SlaveAddress:=ADDRESS;
			MODBUS.MB_Query.FunctionCode:=16#03;
			(* Start query *)
			MODBUS.MB_Query.Read_StartAddress:=addr;
			MODBUS.MB_Query.Read_Quantity:=siz;
			MODBUS.MB_Start:=TRUE;
			sta:=10;
		END_IF

	3:	IF NOT MODBUS.MB_Start THEN
			IF MODBUS.MB_MASTER.MB_Error<>MB_NO_ERROR OR MODBUS.MB_Resp.Error<>0 THEN
				sta:=100;
			ELSE
				(* Read response data *)
				COPY_32SWAP16(ADR(MODBUS.MB_Resp.Data[ 0]),ADR(Data.Vc));
				COPY_32SWAP16(ADR(MODBUS.MB_Resp.Data[ 4]),ADR(Data.Vm));
				COPY_32SWAP16(ADR(MODBUS.MB_Resp.Data[ 6]),ADR(Data.p));
				COPY_32SWAP16(ADR(MODBUS.MB_Resp.Data[ 8]),ADR(Data.t));
				COPY_32SWAP16(ADR(MODBUS.MB_Resp.Data[10]),ADR(Data.Qm));
				COPY_32SWAP16(ADR(MODBUS.MB_Resp.Data[12]),ADR(Data.Qc));
				COPY_32SWAP16(ADR(MODBUS.MB_Resp.Data[14]),ADR(Data.C));
				COPY_32SWAP16(ADR(MODBUS.MB_Resp.Data[16]),ADR(Data.K));
				COPY_32SWAP16(ADR(MODBUS.MB_Resp.Data[18]),ADR(Data.Vcs));
				COPY_32SWAP16(ADR(MODBUS.MB_Resp.Data[22]),ADR(Data.Vms));
				(* Start query *)
				MODBUS.MB_Query.Read_StartAddress:=40052(* <= first *)-40000;
				MODBUS.MB_Query.Read_Quantity:=40055(* <= last *)-40004+1;
				MODBUS.MB_Start:=TRUE;
				sta:=10;
			END_IF
		END_IF

	10:	IF NOT MODBUS.MB_Start THEN
			IF MODBUS.MB_MASTER.MB_Error<>MB_NO_ERROR OR MODBUS.MB_Resp.Error<>0 THEN
				sta:=100;
			ELSE
				(* Read response data *)
				COPY_32SWAP16(ADR(MODBUS.MB_Resp.Data[ 0]),ADR(Data.Vm));
				(*COPY_32SWAP16(ADR(MODBUS.MB_Resp.Data[ 0]),ADR(Data.stat1));
				COPY_32SWAP16(ADR(MODBUS.MB_Resp.Data[ 2]),ADR(Data.stat2));*)
				(* Release MODBUS *)
				MODBUS.MB_Lock:=FALSE;
				(* Update status *)
				Status_Log:=0;
				Status_Vis:=16#20F020;
				sta:=0;
			END_IF
		END_IF

	100: (* === Check MODBUS error *)
		MODBUS.MB_Lock:=FALSE;
		Status_Log:=2;
		Status_Vis:=16#2020F0;
		sta:=0;
*)
ELSE
	sta:=0;
END_CASE
END_FUNCTION_BLOCK
ACTION AddLogData:
Logger.s1:=INSERT('&GASM=',BYTE_TO_STRING(ID),5);
IF ID<10 THEN Logger.s1:=INSERT(Logger.s1,'0',5); END_IF

Logger.s1:=CONCAT(Logger.s1,RAW16TOHEXSTR(ADR(Data.Vb),8));		Logger.s1:=CONCAT(Logger.s1,';');
Logger.s1:=CONCAT(Logger.s1,DWORD_TO_STRING(Data.Vm));			Logger.s1:=CONCAT(Logger.s1,';');
Logger.s1:=CONCAT(Logger.s1,REAL_TO_STRING(Data.P));			Logger.s1:=CONCAT(Logger.s1,';');
Logger.s1:=CONCAT(Logger.s1,REAL_TO_STRING(Data.T));			Logger.s1:=CONCAT(Logger.s1,';');
Logger.s1:=CONCAT(Logger.s1,REAL_TO_STRING(Data.C));			Logger.s1:=CONCAT(Logger.s1,';');
Logger.s1:=CONCAT(Logger.s1,RAW16TOHEXSTR(ADR(Data.Vbs),8));	Logger.s1:=CONCAT(Logger.s1,';');
Logger.s1:=CONCAT(Logger.s1,RAW16TOHEXSTR(ADR(Data.Vb_d_d),8));	Logger.s1:=CONCAT(Logger.s1,';');
Logger.s1:=CONCAT(Logger.s1,RAW16TOHEXSTR(ADR(Data.Vb_d_m),8));	Logger.s1:=CONCAT(Logger.s1,';');
Logger.s1:=CONCAT(Logger.s1,REAL_TO_STRING(Data.Vm_d_d));		Logger.s1:=CONCAT(Logger.s1,';');
Logger.s1:=CONCAT(Logger.s1,REAL_TO_STRING(Data.Q));			Logger.s1:=CONCAT(Logger.s1,';');
Logger.s1:=CONCAT(Logger.s1,REAL_TO_STRING(Data.Qb));			Logger.s1:=CONCAT(Logger.s1,';');
Logger.i1:=REAL_TO_WORD(Data.BC_EVC*10);
Logger.s1:=CONCAT(Logger.s1,WORD_TO_STRING(Logger.i1));			Logger.s1:=CONCAT(Logger.s1,';');

Logger.s1:=CONCAT(Logger.s1,BYTE_TO_STRING(Status_Log));
ADDSTRING(ADR(Logger.TData), ADR(Logger.s1), Logger.TLen);
END_ACTION

(* POU Utils Functions/RAW16TOHEXSTR, ST *)
FUNCTION RAW16TOHEXSTR : STRING(128)
VAR_INPUT
	pData: POINTER TO BYTE;
	DataLen: BYTE;
END_VAR
VAR
	pt: POINTER TO BYTE;
	xl: BYTE;
END_VAR
pt:=ADR(RAW16TOHEXSTR);
xl:=0;

WHILE DataLen>0 AND xl<120 DO

	pData:=pData+1;

	pt^ := (pData^ / 16#10) + 48 + (((pData^ / 16#10)/10)*7);
	pt:=pt+1;
	pt^ := (pData^ AND 16#0F)  + 48 + (((pData^ AND 16#0F)/10)*7);
	pt:=pt+1;

	pData:=pData-1;

	pt^ := (pData^ / 16#10) + 48 + (((pData^ / 16#10)/10)*7);
	pt:=pt+1;
	pt^ := (pData^ AND 16#0F)  + 48 + (((pData^ AND 16#0F)/10)*7);
	pt:=pt+1;

	xl:=xl+4;

	DataLen:=DataLen-2;
	pData:=pData+2;

END_WHILE

pt^:=0;
END_FUNCTION

(* POU PLC_WDT, ST *)
FUNCTION PLC_WDT: DWORD VAR_INPUT dwEvent: DWORD; dwFilter: DWORD; dwOwner: DWORD; END_VAR
LogEv(EL_AlarmStop,EO_SYS,1,10,'Watchdog');
END_FUNCTION

(* POU Utils Functions/RAWTOHEXSTR, ST *)
FUNCTION RAWTOHEXSTR : STRING(128)
VAR_INPUT
	pData: POINTER TO BYTE;
	DataLen: BYTE;
END_VAR
VAR
	pt: POINTER TO BYTE;
	xl: BYTE;
END_VAR
pt:=ADR(RAWTOHEXSTR);

xl:=2;

WHILE DataLen>0 AND xl<128 DO

	pt^ := (pData^ / 16#10) + 48 + (((pData^ / 16#10)/10)*7);
	pt:=pt+1;
	pt^ := (pData^ AND 16#0F)  + 48 + (((pData^ AND 16#0F)/10)*7);
	pt:=pt+1;

	xl:=xl+2;

	DataLen:=DataLen-1;
	pData:=pData+1;

END_WHILE

pt^:=0;
END_FUNCTION

(* POU Utils/RTC_Update, ST *)
FUNCTION RTC_Update : BOOL
VAR
	T: DT;
	TS: STRING;
	TS2: STRING;
	Hour: BYTE;
	Minute: BYTE;
END_VAR
(* Get RTC time *)
T:=SysRtcGetTime(TRUE);
Sys.Time_CT_DT:=T;
(* Calculate variables *)
TS:=DT_TO_STRING(T);
Sys.Time_LogString:=DELETE(STR:=TS, LEN:=3, POS:=1);
TS2:=MID(STR:=TS, LEN:=4, POS:= 4); Sys.Time_Year 	:=STRING_TO_WORD(TS2);
TS2:=MID(STR:=TS, LEN:=2, POS:= 9); Sys.Time_Month	:=STRING_TO_BYTE(TS2);
TS2:=MID(STR:=TS, LEN:=2, POS:=12); Sys.Time_Day  	:=STRING_TO_BYTE(TS2);
Sys.Time_CT_Day:=(32*(Sys.Time_Month-1)+Sys.Time_Day-1);
TS2:=MID(STR:=TS, LEN:=2, POS:=15); Hour			:=STRING_TO_BYTE(TS2);
TS2:=MID(STR:=TS, LEN:=2, POS:=18); Minute		 	:=STRING_TO_BYTE(TS2);
Sys.Time_CT_Quarter:=Hour*4+(Minute/15);
END_FUNCTION

(* POU Utils Functions/TONOF, ST *)
FUNCTION_BLOCK TONOF
VAR_INPUT
	IN		: BOOL;
	PT_ON	: TIME; (* time to pass, before OUT is set *)
	PT_OF	: TIME; (* time to pass, before OUT is reset *)
END_VAR
VAR_OUTPUT
	OUT		: BOOL;
END_VAR
VAR
	timer	: TON;
END_VAR
IF IN<>OUT THEN
	timer(IN:=TRUE,PT:=SEL(IN,PT_OF,PT_ON));
	IF timer.Q THEN OUT:=IN; END_IF
ELSE
	timer(IN:=FALSE);
END_IF
END_FUNCTION_BLOCK

(* Visualisation PLC_VISU
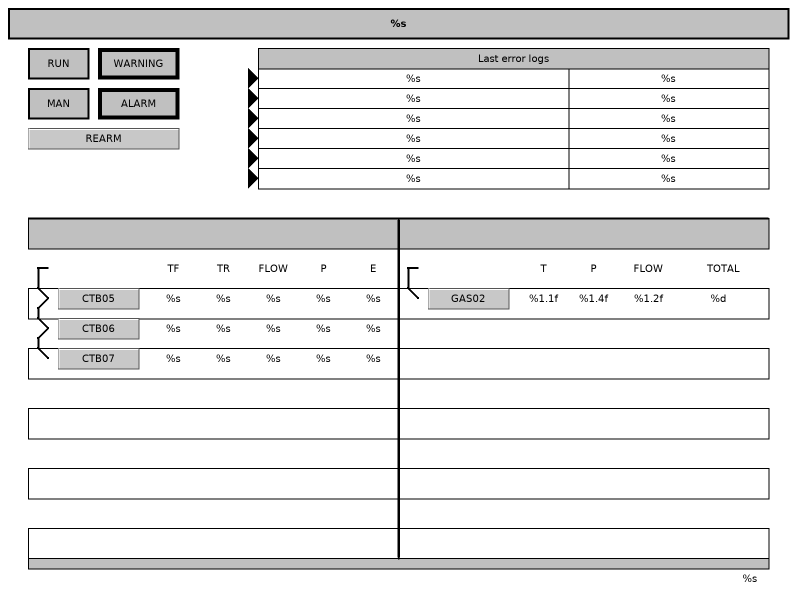
rectangle at (10,10)-(791,41): text "%s"; shows .Plant_NAME
rectangle at (520,570)-(761,591): text "%s"; shows Sys.Time_LogString
rounded rectangle at (30,50)-(91,81): text "RUN"; alarm colour if NOT Mode_Manual; runs INTERN ASSIGN Mode_Manual:=(FALSE)
rounded rectangle at (30,90)-(91,121): text "MAN"; alarm colour if Mode_Manual; runs INTERN ASSIGN Mode_Manual:=(TRUE)
rectangle at (570,70)-(771,91): text "%s"; shows Sys.LastLogs_Msg[0]
polygon at (250,170)-(260,190): invisible if Sys.LastLogs_Idx<>0
rectangle at (570,90)-(771,111): text "%s"; shows Sys.LastLogs_Msg[1]
polygon at (250,70)-(260,90): invisible if Sys.LastLogs_Idx<>1
rectangle at (570,110)-(771,131): text "%s"; shows Sys.LastLogs_Msg[2]
polygon at (250,90)-(260,110): invisible if Sys.LastLogs_Idx<>2
rectangle at (570,130)-(771,151): text "%s"; shows Sys.LastLogs_Msg[3]
polygon at (250,110)-(260,130): invisible if Sys.LastLogs_Idx<>3
rectangle at (570,150)-(771,171): text "%s"; shows Sys.LastLogs_Msg[4]
polygon at (250,130)-(260,150): invisible if Sys.LastLogs_Idx<>4
rectangle at (570,170)-(771,191): text "%s"; shows Sys.LastLogs_Msg[5]
polygon at (250,150)-(260,170): invisible if Sys.LastLogs_Idx<>5
rectangle at (260,70)-(571,91): text "%s"; shows Sys.LastLogs_Dat[0]
rectangle at (260,90)-(571,111): text "%s"; shows Sys.LastLogs_Dat[1]
rectangle at (260,110)-(571,131): text "%s"; shows Sys.LastLogs_Dat[2]
rectangle at (260,130)-(571,151): text "%s"; shows Sys.LastLogs_Dat[3]
rectangle at (260,150)-(571,171): text "%s"; shows Sys.LastLogs_Dat[4]
rectangle at (260,170)-(571,191): text "%s"; shows Sys.LastLogs_Dat[5]
rectangle at (100,90)-(181,121): text "ALARM"; alarm colour if Sys.Alarm; runs INTERN ASSIGN Mode_Manual:=(FALSE)
rectangle at (100,50)-(181,81): text "WARNING"; alarm colour if Sys.Warning; runs INTERN ASSIGN Mode_Manual:=(TRUE)
button at (30,130)-(181,151): text "REARM"; runs INTERN ASSIGN Sys.Alarm:=(FALSE);INTERN ASSIGN Sys.Warning:=(FALSE)
button at (60,290)-(141,311): text "CTB05"
rectangle at (260,50)-(771,71): text "Last error logs"
button at (60,320)-(141,341): text "CTB06"
rectangle at (150,260)-(201,281): text "TF"
rectangle at (250,260)-(301,281): text "FLOW"
rectangle at (300,260)-(351,281): text "P"
rectangle at (350,260)-(401,281): text "E"
rectangle at (200,260)-(251,281): text "TR"
button at (60,350)-(141,371): text "CTB07"
button at (430,290)-(511,311): text "GAS02"
rectangle at (150,290)-(201,311): text "%s"; shows .CTB05.M1.utFTemp.Value
rectangle at (250,290)-(301,311): text "%s"; shows .CTB05.M1.utFlow.Value
rectangle at (300,290)-(351,311): text "%s"; shows .CTB05.M1.utPower.Value
rectangle at (350,290)-(401,311): text "%s"; shows .CTB05.M1.utEnergy.Value
rectangle at (200,290)-(251,311): text "%s"; shows .CTB05.M1.utRTemp.Value
rectangle at (150,320)-(201,341): text "%s"; shows .CTB06.M1.utFTemp.Value
rectangle at (250,320)-(301,341): text "%s"; shows .CTB06.M1.utFlow.Value
rectangle at (300,320)-(351,341): text "%s"; shows .CTB06.M1.utPower.Value
rectangle at (350,320)-(401,341): text "%s"; shows .CTB06.M1.utEnergy.Value
rectangle at (200,320)-(251,341): text "%s"; shows .CTB06.M1.utRTemp.Value
rectangle at (150,350)-(201,371): text "%s"; shows .CTB07.M1.utFTemp.Value
rectangle at (250,350)-(301,371): text "%s"; shows .CTB07.M1.utFlow.Value
rectangle at (300,350)-(351,371): text "%s"; shows .CTB07.M1.utPower.Value
rectangle at (350,350)-(401,371): text "%s"; shows .CTB07.M1.utEnergy.Value
rectangle at (200,350)-(251,371): text "%s"; shows .CTB07.M1.utRTemp.Value
rectangle at (680,260)-(771,281): text "TOTAL"
rectangle at (620,260)-(681,281): text "FLOW"
rectangle at (520,260)-(571,281): text "T"
rectangle at (570,260)-(621,281): text "P"
rectangle at (680,290)-(761,311): text "%d"; shows GAS02.Data.Vm
rectangle at (620,290)-(681,311): text "%1.2f"; shows GAS02.Data.Q
rectangle at (520,290)-(571,311): text "%1.1f"; shows GAS02.Data.T
rectangle at (570,290)-(621,311): text "%1.4f"; shows GAS02.Data.P
11 more shapes without text or variables
6 elements of other kinds (tables, trends, ...) not read
*)
